	END_CASE
ELSE
	_pulseGenerator(IN := TRUE, PT := T#50MS);	
END_IF
END_METHOD

{attribute 'TcRpcEnable' := '1'}
METHOD RaisePropertiesChanged
VAR_INPUT
	Execute : BOOL;
END_VAR
IF Execute THEN	
	DistanceMsg := ' ';
	IdMsg := ' ';
	CustomMsg := ' ';
END_IF
END_METHOD

END_FUNCTION_BLOCK

// ---- PMShared/Hardware/Devices/DistanceSensors/DistanceSensorBase.TcPOU
FUNCTION_BLOCK ABSTRACT DistanceSensorBase EXTENDS TExecution IMPLEMENTS IDevice
VAR_INPUT
END_VAR
VAR_OUTPUT
END_VAR
VAR
	{attribute 'OPC.UA.DA' := '0'}
	_name : STRING;
	{attribute 'OPC.UA.DA' := '0'}
	_deviceID : STRING;					
	{attribute 'OPC.UA.DA' := '0'}
	_family : DeviceFamily;	
	{attribute 'OPC.UA.DA' := '0'}
	_logger : Logger;
	{attribute 'OPC.UA.DA' := '0'}
	_message : StringBuilder;
	{attribute 'OPC.UA.DA' := '0'}
	_distanceSensorConfig : DeviceConfiguration;
END_VAR

PROPERTY DeviceID : STRING
GET
DeviceID := _deviceID;
END_GET
SET
_deviceID := DeviceID;
END_SET
END_PROPERTY

PROPERTY Family : DeviceFamily
GET
Family := _family;
END_GET
SET
_family := Family;
END_SET
END_PROPERTY

PROPERTY Name : STRING
GET
Name := _name;
END_GET
SET
_name := Name;
END_SET
END_PROPERTY

END_FUNCTION_BLOCK

// ---- PMShared/Hardware/Devices/MPPCs/Hamamatsu/C13336/C13336MppcWide.TcPOU
FUNCTION_BLOCK C13336MppcWide EXTENDS C13336Mppc
VAR_INPUT
END_VAR
VAR_OUTPUT
END_VAR
VAR
	{attribute 'OPC.UA.DA' := '0'}
	_config : C13336MppcConfig;
	
	{attribute 'OPC.UA.DA' := '0'}
	_initDevice : BOOL;
	
	{attribute 'OPC.UA.DA.Access' := '0'}
    InputMppcWideStateSignal_1	AT %I* : BOOL;
	
	{attribute 'OPC.UA.DA.Access' := '0'}
    InputMppcWideStateSignal_2	AT %I* : BOOL;
	
	{attribute 'OPC.UA.DA' := '0'}
	_itemInit : INT;
	{attribute 'OPC.UA.DA' := '0'}
	_pulseGeneratorInit : TON;
	
	{attribute 'OPC.UA.DA' := '0'}
	_coeAccess : CoeAccess;
	{attribute 'OPC.UA.DA' := '0'}
	_initConfigSerialCom : BOOL;
	{attribute 'OPC.UA.DA' := '0'}
	_serialCom  : SerialCom(Prefix := Const.START_OF_TEXT, Suffix := Const.CARRIAGE_RETURN);
	{attribute 'OPC.UA.DA' := '0'}
	_refSerialCom : REFERENCE TO SerialCom(Prefix := Const.START_OF_TEXT, Suffix := Const.CARRIAGE_RETURN) := _serialCom;
		
END_VAR

IF NOT _raiseProperties THEN
	GetStateSignals();
END_IF

// Init device
SUPER^.InitDevice();

IF InitConfigSerialCom AND MppcActivate THEN
	THIS^.Status := TExecutionState.Ready;
ELSE
    THIS^.Status := TExecutionState.Error;	
END_IF

IF THIS^.Status = TExecutionState.Ready THEN
	SUPER^(Conf := _config, SerialCom := _serialCom, RefSerialCom := _refSerialCom);
END_IF

IF SUPER^._initDeviceBase THEN	
	IF NOT InitConfigSerialCom THEN
		ConfigureSerialCom();
	ELSIF THIS^.Status = TExecutionState.Ready THEN						
		_refSerialCom(TxBuffer:= HardwareGlobalVariables.TxBufferMppcWide, 
					  RxBuffer:= HardwareGlobalVariables.RxBufferMppcWide);		

		// Start Mppc to off 
		IF NOT _initDevice THEN
			InitDevice();
		END_IF					
	END_IF
END_IF

METHOD ConfigureSerialCom
VAR_INPUT
END_VAR

VAR
	Status: INT;
END_VAR
IF _coeAccess.CoeOperation.Ready THEN
	_logger.Information(_message.Reset().Append('Start configuration com serial').ToString());
END_IF;	

_coeAccess.CoeOperation.Start();
_coeAccess(SerialCommunication := _config.SerialCommunication);
	
IF _coeAccess.CoeOperation.Done THEN
	_coeAccess.SetDone();
	
	_Logger.Information(_message.Reset().
							Append('{').Append(TO_STRING(THIS^.Family)).Append('} : ').
							Append(' - Status : ').Append(TO_STRING(_coeAccess.Status)).ToString());
	InitConfigSerialCom := TRUE;
END_IF
 
IF _coeAccess.CoeOperation.Error THEN	
	_coeAccess.SetError(0);
	
	_Logger.Error(_message.Reset().
							Append('{').Append(TO_STRING(THIS^.Family)).Append('} : ').
							Append(' - Status : ').Append(TO_STRING(_coeAccess.Status)).ToString());
	InitConfigSerialCom := TRUE;
END_IF

THIS^.Status := _coeAccess.Status;
State := _coeAccess.Status;
END_METHOD

METHOD FB_init : BOOL
VAR_INPUT
	bInitRetains : BOOL; // if TRUE, the retain variables are initialized (warm start / cold start)
	bInCopyCode : BOOL;  // if TRUE, the instance afterwards gets moved into the copy code (online change)
	Config : C13336MppcConfig;
END_VAR
IF Config.IsEnabled THEN
	_config := Config;
	
	SUPER^._mppcConfig.Name := Config.Name;
	SUPER^._mppcConfig.DeviceID := Config.DeviceID;
	SUPER^._mppcConfig.IsEnabled := Config.IsEnabled;
	SUPER^._mppcConfig.LogLevel := Config.LogLevel;
	
	SUPER^.Name := Config.Name;
	SUPER^.DeviceID := Config.DeviceID;	
	THIS^.Family := DeviceFamily.MPPC;
		
	_Logger.Information(_message.Reset().Append('Init ').
							Append('{').Append(TO_STRING(THIS^.Family)).Append('} - ').
							Append('{').Append(TO_STRING(Config.Name)).Append('}').ToString());																													
END_IF
END_METHOD

METHOD GetStateSignals
VAR_INPUT
END_VAR
VAR
	{attribute 'OPC.UA.DA' := '0'}
	fibersCollector : STRING;
	{attribute 'OPC.UA.DA' := '0'}
	delimeter : STRING := ';';
	{attribute 'OPC.UA.DA' := '0'}
	stateSignal : STRING;	
	
END_VAR

fibersCollector := CONCAT(TO_STRING(EMppcCollector.WIDE), delimeter);

IF NOT InputMppcWideStateSignal_1 AND NOT InputMppcWideStateSignal_2 THEN
	stateSignal := CONCAT(fibersCollector, TO_STRING(EMppcStateModule.UNRECOVERABLE_ERROR));
ELSIF NOT InputMppcWideStateSignal_1 AND InputMppcWideStateSignal_2 THEN
	stateSignal := CONCAT(fibersCollector, TO_STRING(EMppcStateModule.AWAITING_COOLING_TEMP_STABLE));
ELSIF InputMppcWideStateSignal_1 AND NOT InputMppcWideStateSignal_2 THEN
	stateSignal := CONCAT(fibersCollector, TO_STRING(EMppcStateModule.AWAITING_HIGH_VOLTAGE_POWER_SUPPLY_STABLE));
ELSE
	stateSignal := CONCAT(fibersCollector, TO_STRING(EMppcStateModule.MODULE_OPERATING_NORMAL));
END_IF

IF stateSignal <> SUPER^.StateSignalsMsg THEN	
	SUPER^.StateSignalsMsg := stateSignal;
	SUPER^.GetStateSignals();
END_IF
END_METHOD

PROPERTY InitConfigSerialCom : BOOL
GET
InitConfigSerialCom := _initConfigSerialCom;
END_GET
SET
_initConfigSerialCom := InitConfigSerialCom;
END_SET
END_PROPERTY

METHOD InitDevice
VAR_INPUT
END_VAR
VAR	
END_VAR
IF NOT _initDevice THEN			
	IF _pulseGeneratorInit.Q THEN
		_pulseGeneratorInit(IN := FALSE, PT := T#10MS);
			
		CASE _itemInit OF
			0:  _logger.Information(_message.Reset().
								Append(_config.Name).
								Append(' - Start to on').ToString());		
				_itemInit := 1;
				
			1:  _outputVoltageOn := TRUE;			
				_initDevice := TRUE;
				_itemInit := 0;
		END_CASE
	ELSE
		_pulseGeneratorInit(IN := TRUE, PT := T#500MS);	
	END_IF
END_IF
END_METHOD

END_FUNCTION_BLOCK

// ---- PMShared/Hardware/Devices/MPPCs/Hamamatsu/C13336Mppc.TcPOU
{attribute 'OPC.UA.DA' := '1'}
FUNCTION_BLOCK C13336Mppc EXTENDS MppcBase
VAR_INPUT	
	{attribute 'OPC.UA.DA' := '0'}
	Conf : C13336MppcConfig;
	{attribute 'OPC.UA.DA' := '0'}
	SerialCom  : SerialCom(Prefix := Const.START_OF_TEXT, Suffix := Const.CARRIAGE_RETURN);
	{attribute 'OPC.UA.DA' := '0'}
	RefSerialCom : REFERENCE TO SerialCom(Prefix := Const.START_OF_TEXT, Suffix := Const.CARRIAGE_RETURN) := SerialCom;
	{attribute 'OPC.UA.DA' := '0'}
	MppcActivate : BOOL;
END_VAR
VAR_OUTPUT	
END_VAR
VAR		
	{attribute 'OPC.UA.DA' := '0'}	 
	_isReceived : BOOL;
	
	{attribute 'OPC.UA.DA' := '0'}
	_deliverMessages : INT;
		
	OutputCurrentMsg : STRING(255);
	OutputVoltageMsg : STRING(255);
	OutputVoltageSettingMsg : STRING(255);
	TemperatureMsg : STRING(255);
	SensorTemperatureMsg : STRING(255);
	PowerFctReadMsg : STRING(255);	
	MonitorInfoStatusMsg : STRING(255);
	HighVoltageStatusMsg : STRING(255);	
	TempCorrectionFactorReadMsg : STRING(255);
	FirmwareMsg : STRING(255);
	IdentifierMsg : STRING(255);
	StateSignalsMsg : STRING(255);
	
	{attribute 'OPC.UA.DA' := '0'}
	VoltageStabilityMsg : STRING(255);
	
	{region 'Commands'}
	
	{attribute 'OPC.UA.DA' := '0'}
	_tempCorrectionFactorSetting : BOOL;
	{attribute 'OPC.UA.DA' := '0'}
	_switchTempCompensationMode : BOOL;
	{attribute 'OPC.UA.DA' := '0'}
	_refVoltageTempSetting : BOOL;
	{attribute 'OPC.UA.DA' := '0'}		  
	_powerFctSetting : BOOL;
	{attribute 'OPC.UA.DA' := '0'}			   
	_outputVoltageOn : BOOL;
	{attribute 'OPC.UA.DA' := '0'}		 
	_outputVoltageOff : BOOL;
	{attribute 'OPC.UA.DA' := '0'}
	_powerReset : BOOL;
	{attribute 'OPC.UA.DA' := '0'}
	_customCmd : BOOL;	
	{attribute 'OPC.UA.DA' := '0'}			  		   
	_raiseProperties : BOOL;
	{attribute 'OPC.UA.DA' := '0'}		  
	_powerFctRead : BOOL;
	{attribute 'OPC.UA.DA' := '0'}	
	_overcurrentProtection : BOOL;
	{attribute 'OPC.UA.DA' := '0'}	
	_outputVoltageControl : BOOL;
	{attribute 'OPC.UA.DA' := '0'}	 
	_tempCompensationMode : BOOL;
	{attribute 'OPC.UA.DA' := '0'}			  
	_manageRelays : BOOL;
	{attribute 'OPC.UA.DA' := '0'}
	_ioRelayActivated : BOOL; 
	{attribute 'OPC.UA.DA' := '0'}
	_setOutputVoltage : BOOL;
				   
	{attribute 'OPC.UA.DA' := '0'}
	_collector : STRING;
	{attribute 'OPC.UA.DA' := '0'}
	_fibersCollector : STRING;
	{attribute 'OPC.UA.DA' := '0'}
	_delimeter : STRING := ';';
		 
	{endregion}
		 
	{attribute 'OPC.UA.DA' := '0'}
	_initDeviceBase : BOOL;	
	 
	{attribute 'OPC.UA.DA' := '0'}
	_cmd : STRING;	
	{attribute 'OPC.UA.DA' := '0'}	
	_setRefVoltage : LREAL := 0;
	{attribute 'OPC.UA.DA' := '0'}	
	_setVoltage : LREAL := 0;				
	{attribute 'OPC.UA.DA' := '0'}
	_itemScheduler : INT;		
	{attribute 'OPC.UA.DA' := '0'}
	_itemExecScheduler : INT;
	{attribute 'OPC.UA.DA' := '0'}
	_itemRaisedProperties : INT;
	{attribute 'OPC.UA.DA' := '0'}
	_pulseGenerator : TON;	
			
	{attribute 'OPC.UA.DA' := '0'}
	message : STRING;
	{attribute 'OPC.UA.DA' := '0'}
	tmpMessage : STRING;
	
	{attribute 'OPC.UA.DA' := '0'}
	msgWithoutPrefix : STRING;
	{attribute 'OPC.UA.DA' := '0'}
	suffixDelete : INT := 5;
	{attribute 'OPC.UA.DA' := '0'}
	prefixDelete : INT := 3;
	
	{attribute 'OPC.UA.DA' := '0'}
	_length : INT;
	{attribute 'OPC.UA.DA' := '0'}
	_conv : BOOL;
	{attribute 'OPC.UA.DA' := '0'}
	valConvert : LREAL;		
	
	
	{attribute 'OPC.UA.DA' := '0'}
	strTmp : STRING;
	{attribute 'OPC.UA.DA' := '0'}
	strTmp1 : STRING;
	
END_VAR

IF SerialCom.ErrorSendId <> COMERROR_NOERROR THEN
	RETURN;
END_IF

// Deliver messages
IF RefSerialCom.IsReceived THEN
	IF (Conf.DeviceID = TO_STRING(EMppcCollector.WIDE)) THEN
		_collector := TO_STRING(EMppcCollector.WIDE);
	ELSE
		_collector := TO_STRING(EMppcCollector.NARROW);
	END_IF	
		
	_fibersCollector := CONCAT(_collector, _delimeter);
	
	msgWithoutPrefix := DELETE(RefSerialCom.LastReceivedString, suffixDelete, 0);	
	_length := LEN(msgWithoutPrefix);
	message := DELETE(msgWithoutPrefix, _length - prefixDelete, _length - prefixDelete);

	CASE _deliverMessages OF		
		EFeedbackMsgC13336.MonitorInfoStatusMsg :
		 	MonitorInfoStatusMsg := CONCAT(_fibersCollector, message); 
			VoltageStabilityMsg := CONCAT(_fibersCollector, FindVoltageStability(message)); 
			HighVoltageStatusMsg := CONCAT(_fibersCollector, FindHighVoltageOutput(message));
			
		EFeedbackMsgC13336.OutputCurrentMsg :			
			OutputCurrentMsg := CONCAT(_fibersCollector, ConvertMonitorHexaToCurrent(message));	
			
		EFeedbackMsgC13336.OutputVoltageMsg :
			OutputVoltageMsg := CONCAT(_fibersCollector, ConvertMonitorHexaToVoltage(message));	
			
		EFeedbackMsgC13336.OutputVoltageSettingMsg :			
			tmpMessage := LEFT(RIGHT(message, 8), 4);		
			OutputVoltageSettingMsg := CONCAT(_fibersCollector, ConvertMonitorHexaToVoltage(tmpMessage));		
	
		EFeedbackMsgC13336.TemperatureMsg :
			TemperatureMsg := CONCAT(_fibersCollector, message);
			
		EFeedbackMsgC13336.SensorTemperatureMsg :
			tmpMessage := LEFT(RIGHT(message, 8), 4);
			SensorTemperatureMsg := CONCAT(_fibersCollector, ConvertMonitorHexaToTemperature(tmpMessage));
	
		EFeedbackMsgC13336.PowerFctReadMsg :
			PowerFctReadMsg := CONCAT(_fibersCollector, message);
			
		EFeedbackMsgC13336.TempCorrectionFactorReadMsg :
			TempCorrectionFactorReadMsg := CONCAT(_fibersCollector, message);

		EFeedbackMsgC13336.FirmwareMsg :
			FirmwareMsg := CONCAT(_fibersCollector, message);	
			
		EFeedbackMsgC13336.IdentifierMsg :
			IdentifierMsg := CONCAT(_fibersCollector, message);					
	END_CASE	
END_IF						   							   		
	
TempCorrectionFactorSetting(_tempCorrectionFactorSetting);
SwitchTempCompensationMode(_switchTempCompensationMode, _tempCompensationMode);
RefVoltageTempSetting(_refVoltageTempSetting, _setRefVoltage);
PowerFctSetting(_powerFctSetting, _overcurrentProtection, _outputVoltageControl);
OutputVoltageOn(_outputVoltageOn);
OutputVoltageOff(_outputVoltageOff);
PowerReset(_powerReset);
CustomCommand(_customCmd, _cmd);
RaisePropertiesChanged(_raiseProperties);		
ManageRelays(_manageRelays, _ioRelayActivated);
SetOutputVoltage(_setOutputVoltage, _setVoltage);


IF (NOT _tempCorrectionFactorSetting AND NOT _switchTempCompensationMode AND NOT _refVoltageTempSetting AND NOT _powerFctSetting AND
	NOT _outputVoltageOn AND NOT _outputVoltageOff AND NOT _powerReset AND NOT _raiseProperties AND NOT _manageRelays) THEN
	
	MessageScheduler();	
END_IF

(** Convert Hexa to mA **)
METHOD ConvertMonitorHexaToCurrent : STRING
VAR_INPUT
	Data : STRING;	
END_VAR
VAR
	dataInDec : STRING;
	dataToDint : DINT;
END_VAR
dataInDec := CONCAT('16#', Data);
dataToDint := STRING_TO_DINT(dataInDec);
ConvertMonitorHexaToCurrent := LREAL_TO_FMTSTR(DINT_TO_LREAL(dataToDint) * 0.005194, 3, TRUE);
END_METHOD

(** Convert Hexa to Temperature **)
METHOD ConvertMonitorHexaToTemperature : STRING
VAR_INPUT
	Data : STRING;
END_VAR
VAR
	dataInDec : STRING;
	dataToDint : DINT;
	
	sTmp0 : STRING;
	sTmp1 : STRING;
	sTmp2 : STRING;
	sTemperature : STRING;
END_VAR
dataInDec := CONCAT('16#', Data);
dataToDint := STRING_TO_DINT(dataInDec);

IF dataToDint > 0 THEN
	sTmp0 := LREAL_TO_FMTSTR((DINT_TO_LREAL(dataToDint) * 10000.0) / (1024.0 - DINT_TO_LREAL(dataToDint)) * (1 / 9000.0), 15, FALSE);
	IF STRING_TO_LREAL(sTmp0) > 0 THEN		
		sTmp1 := LREAL_TO_FMTSTR(LN(STRING_TO_LREAL(sTmp0)), 15, FALSE);
		sTmp2 := LREAL_TO_FMTSTR(STRING_TO_LREAL(sTmp1) * (1 / 3410.0) + (1 / 298.15), 15, FALSE);
		sTemperature := LREAL_TO_FMTSTR(1 / STRING_TO_LREAL(sTmp2) - 273.15, 3, FALSE);
	ELSE
		sTemperature := 'NaN';
	END_IF
ELSE
	sTemperature := 'NaN';

END_IF

ConvertMonitorHexaToTemperature := sTemperature;
END_METHOD

(** Convert Hexa to Volt **)
METHOD ConvertMonitorHexaToVoltage : STRING
VAR_INPUT
	Data : STRING;
END_VAR
VAR
	dataInDec : STRING;
	dataToDint : DINT;
END_VAR
dataInDec := CONCAT('16#', Data);
dataToDint := STRING_TO_DINT(dataInDec);
ConvertMonitorHexaToVoltage := LREAL_TO_FMTSTR(DINT_TO_LREAL(dataToDint) * 0.001812, 3, TRUE);
END_METHOD

METHOD ConvertMonitorVoltageToHexa : ARRAY[0..3] OF STRING
VAR_INPUT
	Data : LREAL;
END_VAR
VAR
	dataCoef : STRING;
	dataToDWord : DWORD;	
	
	sMonitorVoltageToHex : STRING;	
	arrayVoltageToHex : ARRAY[0..3] OF STRING;
	
	counter : INT;
	iLenVoltage : INT;
	
	lTmp1 : LREAL;
	lTmp2 : LREAL;
	
	sTmp1 : STRING;
END_VAR
lTmp1 := Data / 0.001812;
lTmp2 := FRAC(lTmp1);
IF lTmp2 < 0.5 THEN
	dataCoef := LREAL_TO_STRING(lTmp1);
ELSE
	dataCoef := LREAL_TO_STRING(lTmp1 + 1);
END_IF

dataToDWord := STRING_TO_DWORD(dataCoef);
sMonitorVoltageToHex := DWORD_TO_HEXSTR(dataToDWord, 4, FALSE);

iLenVoltage := LEN(sMonitorVoltageToHex);
FOR counter := 0 TO iLenVoltage - 1 BY 1 DO
	sTmp1 := MID(sMonitorVoltageToHex, 1, counter + 1);
	arrayVoltageToHex[counter] := BYTE_TO_HEXSTR(F_ToASC(sTmp1), 1, FALSE);
END_FOR;

ConvertMonitorVoltageToHexa := arrayVoltageToHex;
END_METHOD

METHOD ConvertStatusMessage : STRING
VAR_INPUT
	Status : STRING;
END_VAR
VAR
	voltageOutputMessage : BOOL;

	tmp : UINT;		
END_VAR
tmp := STRING_TO_UINT(RIGHT(Status, 1));

voltageOutputMessage := UINT_TO_BOOL(tmp);

IF voltageOutputMessage THEN
	ConvertStatusMessage := 'ON'; 	
ELSE
	ConvertStatusMessage := 'OFF';
END_IF
END_METHOD

{attribute 'TcRpcEnable' := '1'}
(** Custom command **)
METHOD CustomCommand 
VAR_INPUT
	Execute : BOOL;
	Cmd : STRING;
END_VAR
IF Execute THEN
	_logger.Information(_message.Reset().
								Append(Conf.Name).
								Append(' - Custom command : ').
								Append(Cmd).ToString());	
	_deliverMessages := EFeedbackMsgC13336.CustomMsg;														
	SerialCom.Send(Cmd);	
	_customCmd := FALSE;
END_IF
END_METHOD

METHOD FindHighVoltageOutput : STRING
VAR_INPUT
	message : STRING;
END_VAR
VAR
	{attribute 'OPC.UA.DA' := '0'}	
	_monitorHighVoltageStatus : STRING(255);			
	{attribute 'OPC.UA.DA' := '0'}
	statusMessageBin : STRING;
	{attribute 'OPC.UA.DA' := '0'}
	messageToBin : STRING;
	{attribute 'OPC.UA.DA' := '0'}		
	mask : STRING := '16#1';
	{attribute 'OPC.UA.DA' := '0'}
	status : WORD;
	{attribute 'OPC.UA.DA' := '0'}
	statusMsg : WORD;
END_VAR
statusMsg := STRING_TO_WORD(CONCAT('16#', LEFT(message, 4)));
statusMessageBin := WORD_TO_BINSTR(statusMsg, 16);

status := STRING_TO_WORD(statusMessageBin) AND STRING_TO_WORD(mask);

IF status = 0 THEN
	_monitorHighVoltageStatus := 'OFF';
ELSE
	_monitorHighVoltageStatus := 'ON';
END_IF

FindHighVoltageOutput := _monitorHighVoltageStatus;
END_METHOD

METHOD FindVoltageStability : STRING
VAR_INPUT
	message : STRING;
END_VAR
VAR
	{attribute 'OPC.UA.DA' := '0'}	
	_monitorInfoStatus : STRING(255);		
	{attribute 'OPC.UA.DA' := '0'}
	one : WORD := 1;
	{attribute 'OPC.UA.DA' := '0'}
	isolStatus : DWORD;
	{attribute 'OPC.UA.DA' := '0'}
	statusMessageBin : STRING;
	{attribute 'OPC.UA.DA' := '0'}
	messageToBin : STRING;
	{attribute 'OPC.UA.DA' := '0'}
	valueStatus : WORD;
	{attribute 'OPC.UA.DA' := '0'}		
	mask : STRING := '16#4000';
	{attribute 'OPC.UA.DA' := '0'}
	status : WORD;
	{attribute 'OPC.UA.DA' := '0'}
	statusMsg : WORD;
	
END_VAR

statusMsg := STRING_TO_WORD(CONCAT('16#', LEFT(message, 4)));
statusMessageBin := WORD_TO_BINSTR(statusMsg, 16);

status := STRING_TO_WORD(statusMessageBin) AND STRING_TO_WORD(mask);
valueStatus := SHR(status, 14);


IF valueStatus = 0 THEN
	_monitorInfoStatus := 'Unstable';
ELSE
	_monitorInfoStatus := 'Stable';
END_IF

FindVoltageStability := _monitorInfoStatus;
END_METHOD

METHOD GetFirmware
VAR_INPUT
END_VAR
VAR
	// 'HFI'
	cmdArray : ARRAY[0..7] OF BYTE := [16#02, 16#48, 16#46, 16#49, 16#03, 16#44, 16#43, 16#0D];
END_VAR
_deliverMessages := EFeedbackMsgC13336.FirmwareMsg;
SerialCom.Send8B(cmdArray);
END_METHOD

METHOD GetIdentifier
VAR_INPUT
END_VAR
VAR
	// 'HGN'
	cmdArray : ARRAY[0..7] OF BYTE := [16#02, 16#48, 16#47, 16#4F, 16#03, 16#45, 16#32, 16#0D]; 
END_VAR
 _deliverMessages := EFeedbackMsgC13336.IdentifierMsg;
SerialCom.Send8B(cmdArray);
END_METHOD

METHOD GetMonitorInfoStatus
VAR_INPUT
END_VAR
VAR
	// 'HPO'
	cmdArray : ARRAY[0..7] OF BYTE := [16#02, 16#48, 16#50, 16#4F, 16#03, 16#45, 16#43, 16#0D];
END_VAR
_deliverMessages := EFeedbackMsgC13336.MonitorInfoStatusMsg;
SerialCom.Send8B(cmdArray);
END_METHOD

METHOD GetOutputCurrent
VAR_INPUT
END_VAR
VAR
	// 'HGC'
	cmdArray : ARRAY[0..7] OF BYTE := [16#02, 16#48, 16#47, 16#43, 16#03, 16#44, 16#37, 16#0D]; 
END_VAR
_deliverMessages := EFeedbackMsgC13336.OutputCurrentMsg;
SerialCom.Send8B(cmdArray);
END_METHOD

METHOD GetOutputVoltage
VAR_INPUT
END_VAR
VAR
	// 'HGV'
	cmdArray : ARRAY[0..7] OF BYTE := [16#02, 16#48, 16#47, 16#56, 16#03, 16#45, 16#41, 16#0D]; 
END_VAR
_deliverMessages := EFeedbackMsgC13336.OutputVoltageMsg;
SerialCom.Send8B(cmdArray);
END_METHOD

METHOD GetOutputVoltageSetting
VAR_INPUT
END_VAR
VAR
	// 'HRT'
	cmdArray : ARRAY[0..7] OF BYTE := [16#02, 16#48, 16#52, 16#54, 16#03, 16#46, 16#33, 16#0D]; 
END_VAR
_deliverMessages := EFeedbackMsgC13336.OutputVoltageSettingMsg;
SerialCom.Send8B(cmdArray);
END_METHOD

METHOD GetSensorTemperature
VAR_INPUT
END_VAR
VAR
	// 'TGV'
	cmdArray : ARRAY[0..7] OF BYTE := [16#02, 16#54, 16#47, 16#56, 16#03, 16#46, 16#36, 16#0D]; 
END_VAR
_deliverMessages := EFeedbackMsgC13336.SensorTemperatureMsg;
SerialCom.Send8B(cmdArray);
END_METHOD

METHOD GetStateSignals
VAR_INPUT
END_VAR
_deliverMessages := EFeedbackMsgC13336.StateSignalsMsg;
END_METHOD

METHOD GetStatus
VAR
	// 'HGS'
	cmdArray : ARRAY[0..7] OF BYTE := [16#02, 16#48, 16#47, 16#53, 16#03, 16#45, 16#37, 16#0D]; 
END_VAR
_deliverMessages := EFeedbackMsgC13336.StatusMsg;
SerialCom.Send8B(cmdArray);
END_METHOD

METHOD GetTemperature
VAR_INPUT
END_VAR
VAR
	// 'HGT'
	cmdArray : ARRAY[0..7] OF BYTE := [16#02, 16#48, 16#47, 16#54, 16#03, 16#45, 16#38, 16#0D]; 
END_VAR
_deliverMessages := EFeedbackMsgC13336.TemperatureMsg;
SerialCom.Send8B(cmdArray);
END_METHOD

METHOD InitDevice
VAR_INPUT
END_VAR
IF NOT _initDeviceBase THEN	
	_logger.Information(_message.Reset().
								Append(Conf.Name).
								Append(' - Activates relays').ToString());
		
	ManageRelays(TRUE, TRUE);			
	_initDeviceBase := TRUE;	
END_IF
END_METHOD

METHOD ManageRelays
VAR_INPUT
	Execute : BOOL;
	IoRelay : BOOL;
END_VAR
IF Execute THEN
	_logger.Information(_message.Reset().
								Append('MPPCs relay: ').
								Append(BOOL_TO_STRING(IoRelay)).ToString());	

	// Physically activates relay			
	MppcActivate := IoRelay;
	
	_manageRelays := FALSE;
END_IF
END_METHOD

METHOD MessageScheduler
VAR_INPUT
END_VAR
IF _pulseGenerator.Q THEN
	_pulseGenerator(IN := FALSE, PT := T#10MS);
		
	CASE _itemScheduler OF		
		0: GetOutputCurrent();
			_itemScheduler := 1;
				
		1: GetOutputVoltage();
			_itemScheduler := 2;
			
		2: GetMonitorInfoStatus();
			_itemScheduler := 3;
			
		3: GetSensorTemperature();
			_itemScheduler := 0;
	END_CASE
ELSE
	_pulseGenerator(IN := TRUE, PT := T#200MS);	
END_IF
END_METHOD

{attribute 'TcRpcEnable' := '1'}
METHOD OutputVoltageOff
VAR_INPUT
	Execute : BOOL;
END_VAR
VAR	
	// 'HOF'
	cmdArray : ARRAY[0..7] OF BYTE := [16#02, 16#48, 16#4F, 16#46, 16#03, 16#45, 16#32, 16#0D]; 
END_VAR
IF Execute THEN		
	_outputVoltageOff := TRUE;
	
	IF _pulseGenerator.Q THEN
		_pulseGenerator(IN := FALSE, PT := T#10MS);
		
		CASE _itemExecScheduler OF		
			0:  _logger.Information(_message.Reset().
								Append(Conf.Name).
								Append(' - OutputVoltageOff').ToString());
				SerialCom.Send8B(cmdArray);   
				_itemExecScheduler := 1;
				
			1: GetStatus(); 
				_outputVoltageOff := FALSE;
				_itemExecScheduler := 0;
		
		END_CASE	
	ELSE
		_pulseGenerator(IN := TRUE, PT := T#200MS);	
	END_IF									
END_IF
END_METHOD

{attribute 'TcRpcEnable' := '1'}
METHOD OutputVoltageOn
VAR_INPUT
	Execute : BOOL;
END_VAR
VAR
	// 'HON'
	cmdArray : ARRAY[0..7] OF BYTE := [16#02, 16#48, 16#4F, 16#4E, 16#03, 16#45, 16#41, 16#0D]; 
END_VAR
IF Execute THEN		
	_outputVoltageOn := TRUE;
	
	IF _pulseGenerator.Q THEN
		_pulseGenerator(IN := FALSE, PT := T#10MS);
		
		CASE _itemExecScheduler OF		
			0:  _logger.Information(_message.Reset().
								Append(Conf.Name).
								Append(' - OutputVoltageOn').ToString());
				SerialCom.Send8B(cmdArray);   
				_itemExecScheduler := 0;
				_outputVoltageOn := FALSE;
				
			1: GetStatus(); 
				_outputVoltageOn := FALSE;
				_itemExecScheduler := 0;
		
		END_CASE	
	ELSE
		_pulseGenerator(IN := TRUE, PT := T#2000MS);	
	END_IF									
END_IF
END_METHOD

METHOD PowerFctRead
VAR_INPUT	
END_VAR
VAR
	// 'HRC'
	cmdArray : ARRAY[0..7] OF BYTE := [16#02, 16#48, 16#52, 16#43, 16#03, 16#45, 16#32, 16#0D]; 
END_VAR
_deliverMessages := EFeedbackMsgC13336.PowerFctReadMSg;
SerialCom.Send8B(cmdArray);
END_METHOD

{attribute 'TcRpcEnable' := '1'}
METHOD PowerFctSetting
VAR_INPUT
	Execute : BOOL;
	OvercurrentProtection : BOOL;
	OutputVoltageControl : BOOL;
END_VAR
VAR
	// 'HSC'
	cmdArray : ARRAY[0..11] OF BYTE; 
	data : BYTE := 16#32;
	checksum : BYTE;
END_VAR
IF Execute THEN
	_logger.Information(_message.Reset().
								Append(Conf.Name).
								Append(' - PowerFctSetting').ToString());		

	IF OvercurrentProtection AND OutputVoltageControl THEN 
		data := 16#33;
		checksum := 16#36;
	ELSIF OvercurrentProtection AND NOT OutputVoltageControl THEN
		data := 16#31;
		checksum := 16#34;
	ELSIF NOT OvercurrentProtection AND OutputVoltageControl THEN
		data := 16#32;
		checksum := 16#35;
	ELSE
		data := 16#30;
		checksum := 16#33;	
	END_IF	
	
	cmdArray[0] := 16#02;
	cmdArray[1] := 16#48; 
	cmdArray[2] := 16#53; 
	cmdArray[3] := 16#43; 
	cmdArray[4] := 16#30; 
	cmdArray[5] := 16#30; 
	cmdArray[6] := 16#30; 
	cmdArray[7] := data;	
	cmdArray[8] := 16#03; 
	cmdArray[9] := 16#41; 
	cmdArray[10] := checksum; 
	cmdArray[11] := 16#0D; 
										
	SerialCom.Send12B(cmdArray);
	_powerFctSetting := FALSE;
END_IF
END_METHOD

{attribute 'TcRpcEnable' := '1'}
METHOD PowerReset
VAR_INPUT
	Execute : BOOL;
END_VAR
VAR
	// 'HRE'
	cmdArray : ARRAY[0..7] OF BYTE := [16#02, 16#48, 16#52, 16#45, 16#03, 16#45, 16#34, 16#0D]; 
END_VAR
IF Execute THEN		
	_powerReset := TRUE;
	
	IF _pulseGenerator.Q THEN
		_pulseGenerator(IN := FALSE, PT := T#10MS);
		
		CASE _itemExecScheduler OF		
			0:  _logger.Information(_message.Reset().
								Append(Conf.Name).
								Append(' - PowerReset').ToString());
				SerialCom.Send8B(cmdArray);   
				_itemExecScheduler := 2;				
				
			1: GetStatus(); 
				_itemExecScheduler := 2;
				
			2:	_powerReset := FALSE;
				_itemExecScheduler := 0;
		
		END_CASE	
	ELSE
		_pulseGenerator(IN := TRUE, PT := T#500MS);	
	END_IF									
END_IF
END_METHOD

{attribute 'TcRpcEnable' := '1'}
METHOD RaisePropertiesChanged
VAR_INPUT
	Execute : BOOL;
END_VAR

(*
Ajouter fonction pour remonter les états des 2 IOs quand C# en fait la demande.
La même chose avec LE On/off où l'info n'est pas remontée vu qu'elle n'a pas changé
*)
IF Execute THEN	
	_raiseProperties := TRUE;
	
	IF _pulseGenerator.Q THEN
		_pulseGenerator(IN := FALSE, PT := T#10MS);
	
		CASE _itemRaisedProperties OF		
			0:  //OutputCurrentMsg := ' ';	
				//OutputVoltageMsg := ' ';			    		   			    		   
			    //SensorTemperatureMsg := ' ';			    
				OutputVoltageSettingMsg := ' ';	
			    StateSignalsMsg := ' ';	
			    			    
			    TemperatureMsg := ' ';
			    FirmwareMsg := ' ';
			    TempCorrectionFactorReadMsg := ' ';				   
   			    HighVoltageStatusMsg := ' ';	
                IdentifierMsg := ' ';
			    PowerFctReadMsg := ' ';		   
			   
				_itemRaisedProperties := 10;													

			10:  GetOutputVoltageSetting();
				_itemRaisedProperties := 11;			
				
			11: GetStateSignals();
				_itemRaisedProperties := 12;
								
			12: _logger.Information(_message.Reset().Append(Conf.Name).
													 Append(' - RaisePropertiesChanged').ToString());
				_raiseProperties := FALSE;
				_itemRaisedProperties := 0;
				
			(* Not necessary for the moment *)			
			30: GetOutputCurrent();
				_itemRaisedProperties := 31;

			31: GetOutputVoltage();
				_itemRaisedProperties := 32;						
																				
			32: GetSensorTemperature();
				_itemRaisedProperties := 33;
			
			33: GetMonitorInfoStatus();
				_itemRaisedProperties := 34;
								
			34: GetFirmware();
				_itemRaisedProperties := 35;
				
			35: TempCorrectionFactorRead();
				_itemRaisedProperties := 36;
				
			36: GetTemperature();
				_itemRaisedProperties := 37;
				
			37: PowerFctRead();
				_itemRaisedProperties := 38;
				
			38: GetIdentifier();
				_itemRaisedProperties := 0;
									
		END_CASE
	
	ELSE
		_pulseGenerator(IN := TRUE, PT := T#500MS);	
	END_IF
END_IF
END_METHOD

{attribute 'TcRpcEnable' := '1'}
METHOD RefVoltageTempSetting
VAR_INPUT
	Execute    : BOOL;
	RefVoltage : LREAL;
END_VAR
VAR
	convertToString : STRING;

	refVoltatgeToArray : ARRAY[0..3] OF STRING; 	

	// 'HBV'
	cmdArray : ARRAY[0..11] OF BYTE; // := [2, 48, 66, 86, 55, 53, 69, 66, 3, 50, 67, 13];
END_VAR
IF Execute THEN
	_logger.Information(_message.Reset().
								Append(Conf.Name).
								Append(' - RefVoltageTempSetting').ToString());	

	refVoltatgeToArray := ConvertMonitorVoltageToHexa(RefVoltage);	

	cmdArray[0] := 16#02;
	cmdArray[1] := 16#30; //48;
	cmdArray[2] := 16#42; //66;
	cmdArray[3] := 16#56; //86;	
	cmdArray[4] := STRING_TO_BYTE(refVoltatgeToArray[0]);
	cmdArray[5] := STRING_TO_BYTE(refVoltatgeToArray[1]);
	cmdArray[6] := STRING_TO_BYTE(refVoltatgeToArray[2]);
	cmdArray[7] := STRING_TO_BYTE(refVoltatgeToArray[3]);	
	cmdArray[8] :=16#03;
	cmdArray[9] := 16#32; //50;
	cmdArray[10] := 16#43; //67;
	cmdArray[11] := 16#0D; //13;
				
	SerialCom.Send12B(cmdArray);
	_refVoltageTempSetting := FALSE;
END_IF
END_METHOD

{attribute 'TcRpcEnable' := '1'}
METHOD SetOutputVoltage
VAR_INPUT
	Execute : BOOL;
	SetVoltage : LREAL;
END_VAR
VAR
	convertToString : STRING;
	setVoltatgeToArrayToHex : ARRAY[0..3] OF STRING; 	

	// 'HST'
	cmdArray : ARRAY[0..31] OF BYTE; 
	
	voltageChecksum : DINT;
	counter : INT;
	
	sPartOfChecksum : STRING := '16#4B4'; // Part of checksum, without voltage value (in hex)	
	wSumVoltageValueToHex : WORD;
	wChecksumTotalToDec : WORD;
	sChecksumTotalToHex : STRING;
	ArrayChecksum : ARRAY[0..MAX_STRING_LENGTH] OF BYTE;
	
	iLenCheksum : INT;
	lastByteChecksum : BYTE;
	secondLastByteChecksum : BYTE;
	
	sLastByteChecksum : STRING;
	sSecondLastByteChecksum : STRING;	
	
	sLastByteChecksumHex : STRING;
	sSecondLastByteChecksumHex : STRING;
	
END_VAR
IF Execute THEN
	_logger.Information(_message.Reset().
								Append(Conf.Name).
								Append(' - Set Output Voltage').ToString());	

	setVoltatgeToArrayToHex := ConvertMonitorVoltageToHexa(SetVoltage);	

	(** Checksum **)
	// Add voltage value and convert it to decimal  
	FOR counter := 0 TO 3 BY 1 DO
		IF counter = 0 THEN
			wSumVoltageValueToHex := STRING_TO_WORD(CONCAT('16#', setVoltatgeToArrayToHex[counter]));
		ELSE
			wSumVoltageValueToHex := wSumVoltageValueToHex + STRING_TO_WORD(CONCAT('16#', setVoltatgeToArrayToHex[counter]));	
		END_IF					
	END_FOR;	
	
	wChecksumTotalToDec := STRING_TO_WORD(sPartOfChecksum) + wSumVoltageValueToHex;
	sChecksumTotalToHex := DWORD_TO_HEXSTR(wChecksumTotalToDec, 1, FALSE);		
	
	ArrayChecksum := MAXSTRING_TO_BYTEARR(sChecksumTotalToHex);
	iLenCheksum := LEN(sChecksumTotalToHex);	
	
	sSecondLastByteChecksum := MID(sChecksumTotalToHex, 1, iLenCheksum-1);
	sSecondLastByteChecksumHex := BYTE_TO_HEXSTR(F_ToASC(sSecondLastByteChecksum), 1, FALSE);
	sLastByteChecksum := MID(sChecksumTotalToHex, 1, iLenCheksum);	
	sLastByteChecksum :=  BYTE_TO_HEXSTR(F_ToASC(sLastByteChecksum), 1, FALSE);
		
	cmdArray[0] := 16#02;
	cmdArray[1] := 16#48; //72;
	cmdArray[2] := 16#53; //83;
	cmdArray[3] := 16#54; //84;
	cmdArray[4] := 16#30; //48;
	cmdArray[5] := 16#30; //48;
	cmdArray[6] := 16#30; //48;
	cmdArray[7] := 16#30; //48;
	cmdArray[8] := 16#30; //48;
	cmdArray[9] := 16#30; //48;
	cmdArray[10] := 16#30; //48;
	cmdArray[11] := 16#30; //48;
	cmdArray[12] := 16#30; //48;
	cmdArray[13] := 16#30; //48;
	cmdArray[14] := 16#30; //48;
	cmdArray[15] := 16#30; //48;
	cmdArray[16] := 16#30; //48;
	cmdArray[17] := 16#30; //48;
	cmdArray[18] := 16#30; //48;
	cmdArray[19] := 16#30; //48;	
	cmdArray[20] := STRING_TO_BYTE(CONCAT('16#', setVoltatgeToArrayToHex[0]));
	cmdArray[21] := STRING_TO_BYTE(CONCAT('16#', setVoltatgeToArrayToHex[1]));
	cmdArray[22] := STRING_TO_BYTE(CONCAT('16#', setVoltatgeToArrayToHex[2]));
	cmdArray[23] := STRING_TO_BYTE(CONCAT('16#', setVoltatgeToArrayToHex[3]));
	cmdArray[24] := 16#30; //48;
	cmdArray[25] := 16#30; //48;
	cmdArray[26] := 16#30; //48;
	cmdArray[27] := 16#30; //48;		
	cmdArray[28] := 16#03;
	cmdArray[29] := STRING_TO_BYTE(CONCAT('16#', sSecondLastByteChecksumHex)); // 16#38 -> 56;
	cmdArray[30] := STRING_TO_BYTE(CONCAT('16#', slastByteChecksum)); // 16#42 -> 66;
	cmdArray[31] := 16#0D; //13;
				
	SerialCom.Send32B(cmdArray);
	_setOutputVoltage := FALSE;
END_IF
END_METHOD

{attribute 'TcRpcEnable' := '1'}
METHOD SwitchTempCompensationMode
VAR_INPUT
	Execute : BOOL;
	TempCompensationMode : BOOL; //0: Disable, 1: Enable
END_VAR
VAR
	// 'HCM'
	cmdArray : ARRAY[0..8] OF BYTE; 
	compensationMode : BYTE;
	mode : STRING;
END_VAR
IF Execute THEN
	IF TempCompensationMode THEN
		compensationMode := 49;
		mode := 'Enable';
	ELSE
		compensationMode := 48;
		mode := 'Disable';
	END_IF	
	
	_logger.Information(_message.Reset().Append(Conf.Name).
										 Append(' - SwitchTempCompensationMode: ').
										 Append(mode).ToString());
	
	cmdArray[0] := 16#02;
	cmdArray[1] := 16#48;//72;
	cmdArray[2] := 16#43;//67;
	cmdArray[3] := 16#4D;//77;	
	cmdArray[4] := compensationMode;
	cmdArray[5] := 16#03;
	cmdArray[6] := 16#30;//48;
	cmdArray[7] := 16#45;//69;	
	cmdArray[8] := 16#0D;//13;
							
	SerialCom.Send9B(cmdArray);
	_switchTempCompensationMode := FALSE;
END_IF
END_METHOD

METHOD TempCorrectionFactorRead
VAR_INPUT
END_VAR
VAR
	// 'HRT'
	cmdArray : ARRAY[0..7] OF BYTE := [16#02, 16#30, 16#52, 16#54, 16#03, 16#46, 16#33, 16#0D];
END_VAR
_deliverMessages := EFeedbackMsgC13336.TempCorrectionFactorReadMsg;
SerialCom.Send8B(cmdArray);
END_METHOD

{attribute 'TcRpcEnable' := '1'}
METHOD TempCorrectionFactorSetting
VAR_INPUT
	Execute : BOOL;
END_VAR
VAR
	// 'HST'
	cmdArray : ARRAY[0..7] OF BYTE := [16#02, 16#30, 16#53, 16#54, 16#03, 16#46, 16#34, 16#0D];
END_VAR
IF Execute THEN
	_logger.Information(_message.Reset().
								Append(Conf.Name).
								Append(' - TempCorrectionFactorSetting').ToString());								
	SerialCom.Send8B(cmdArray);
	_tempCorrectionFactorSetting := FALSE;
END_IF
END_METHOD

END_FUNCTION_BLOCK

// ---- PMShared/Hardware/Devices/MPPCs/MppcBase.TcPOU
FUNCTION_BLOCK ABSTRACT MppcBase EXTENDS TExecution IMPLEMENTS IDevice
VAR_INPUT
END_VAR
VAR_OUTPUT
END_VAR
VAR
	{attribute 'OPC.UA.DA' := '0'}
	_name : STRING;
	{attribute 'OPC.UA.DA' := '0'}
	_deviceID : STRING;					
	{attribute 'OPC.UA.DA' := '0'}
	_family : DeviceFamily;	
	{attribute 'OPC.UA.DA' := '0'}	
	_logger : Logger;
	{attribute 'OPC.UA.DA' := '0'}
	_message : StringBuilder;
	{attribute 'OPC.UA.DA' := '0'}
	_mppcConfig : DeviceConfiguration;
	

END_VAR

PROPERTY DeviceID : STRING
GET
DeviceID := _deviceID;
END_GET
SET
_deviceID := DeviceID;
END_SET
END_PROPERTY

PROPERTY Family : DeviceFamily
GET
Family := _family;
END_GET
SET
_family := Family;
END_SET
END_PROPERTY

PROPERTY Name : STRING
GET
Name := _name;
END_GET
SET
_name := Name;
END_SET
END_PROPERTY

END_FUNCTION_BLOCK

// ---- PMShared/Hardware/Devices/MPPCs/Hamamatsu/C13336/C13366MppcNarrow.TcPOU
FUNCTION_BLOCK C13366MppcNarrow EXTENDS C13336Mppc
VAR_INPUT
END_VAR
VAR_OUTPUT
END_VAR
VAR
	{attribute 'OPC.UA.DA' := '0'}
	_config : C13336MppcConfig;
	
	{attribute 'OPC.UA.DA' := '0'}
	_initDevice : BOOL;
	
	{attribute 'OPC.UA.DA.Access' := '0'}
    InputMppcNarrowStateSignal_1	AT %I* : BOOL;
	
	{attribute 'OPC.UA.DA.Access' := '0'}
    InputMppcNarrowStateSignal_2	AT %I* : BOOL;
	
	{attribute 'OPC.UA.DA' := '0'}
	_itemInit : INT;
	{attribute 'OPC.UA.DA' := '0'}
	_pulseGeneratorInit : TON;
	
	{attribute 'OPC.UA.DA' := '0'}
	_coeAccess : CoeAccess;
	{attribute 'OPC.UA.DA' := '0'}
	_initConfigSerialCom : BOOL;
	{attribute 'OPC.UA.DA' := '0'}
	_serialCom  : SerialCom(Prefix := Const.START_OF_TEXT, Suffix := Const.CARRIAGE_RETURN);
	{attribute 'OPC.UA.DA' := '0'}
	_refSerialCom : REFERENCE TO SerialCom(Prefix := Const.START_OF_TEXT, Suffix := Const.CARRIAGE_RETURN) := _serialCom;
END_VAR

IF NOT _raiseProperties THEN
	GetStateSignals();
END_IF

// Init device
SUPER^.InitDevice();

IF InitConfigSerialCom AND MppcActivate THEN
	THIS^.Status := TExecutionState.Ready;
ELSE
    THIS^.Status := TExecutionState.Error;	
END_IF

IF THIS^.Status = TExecutionState.Ready THEN
	SUPER^(Conf := _config, SerialCom := _serialCom, RefSerialCom := _refSerialCom);
END_IF

IF SUPER^._initDeviceBase THEN
	IF NOT InitConfigSerialCom THEN
		ConfigureSerialCom();
	ELSIF THIS^.Status = TExecutionState.Ready THEN			
		_refSerialCom(TxBuffer:= HardwareGlobalVariables.TxBufferMppcNarrow, 
					  RxBuffer:= HardwareGlobalVariables.RxBufferMppcNarrow);
		
		// Start Mppc to off 
		IF NOT _initDevice THEN
			InitDevice();
		END_IF				
	END_IF
END_IF

METHOD ConfigureSerialCom
VAR_INPUT
END_VAR

VAR
	Status: INT;
END_VAR
IF _coeAccess.CoeOperation.Ready THEN
	_logger.Information(_message.Reset().Append('Start configuration com serial').ToString());
END_IF;	

_coeAccess.CoeOperation.Start();
_coeAccess(SerialCommunication := _config.SerialCommunication);
	
IF _coeAccess.CoeOperation.Done THEN
	_coeAccess.SetDone();
	
	_Logger.Information(_message.Reset().
							Append('{').Append(TO_STRING(THIS^.Family)).Append('} : ').
							Append(' - Status : ').Append(TO_STRING(_coeAccess.Status)).ToString());
	InitConfigSerialCom := TRUE;
END_IF
 
IF _coeAccess.CoeOperation.Error THEN	
	_coeAccess.SetError(0);
	
	_Logger.Error(_message.Reset().
							Append('{').Append(TO_STRING(THIS^.Family)).Append('} : ').
							Append(' - Status : ').Append(TO_STRING(_coeAccess.Status)).ToString());
	InitConfigSerialCom := TRUE;
END_IF

THIS^.Status := _coeAccess.Status;
State := _coeAccess.Status;
END_METHOD

METHOD FB_init : BOOL
VAR_INPUT
	bInitRetains : BOOL; // if TRUE, the retain variables are initialized (warm start / cold start)
	bInCopyCode : BOOL;  // if TRUE, the instance afterwards gets moved into the copy code (online change)
	Config : C13336MppcConfig;
END_VAR
IF Config.IsEnabled THEN
	_config := Config;
	
	SUPER^._mppcConfig.Name := Config.Name;
	SUPER^._mppcConfig.DeviceID := Config.DeviceID;
	SUPER^._mppcConfig.IsEnabled := Config.IsEnabled;
	SUPER^._mppcConfig.LogLevel := Config.LogLevel;
	
	SUPER^.Name := Config.Name;
	SUPER^.DeviceID := Config.DeviceID;	
	THIS^.Family := DeviceFamily.MPPC;
		
	_Logger.Information(_message.Reset().Append('Init ').
							Append('{').Append(TO_STRING(THIS^.Family)).Append('} - ').
							Append('{').Append(TO_STRING(Config.Name)).Append('}').ToString());																													
END_IF
END_METHOD

METHOD GetStateSignals
VAR_INPUT
END_VAR
VAR
	{attribute 'OPC.UA.DA' := '0'}
	fibersCollector : STRING;
	{attribute 'OPC.UA.DA' := '0'}
	delimeter : STRING := ';';
	{attribute 'OPC.UA.DA' := '0'}
	stateSignal : STRING;
END_VAR

fibersCollector := CONCAT(TO_STRING(EMppcCollector.NARROW), delimeter);

IF NOT InputMppcNarrowStateSignal_1 AND NOT InputMppcNarrowStateSignal_2 THEN
	stateSignal := CONCAT(fibersCollector, TO_STRING(EMppcStateModule.UNRECOVERABLE_ERROR));
ELSIF NOT InputMppcNarrowStateSignal_1 AND InputMppcNarrowStateSignal_2 THEN
	stateSignal := CONCAT(fibersCollector, TO_STRING(EMppcStateModule.AWAITING_COOLING_TEMP_STABLE));
ELSIF InputMppcNarrowStateSignal_1 AND NOT InputMppcNarrowStateSignal_2 THEN
	stateSignal := CONCAT(fibersCollector, TO_STRING(EMppcStateModule.AWAITING_HIGH_VOLTAGE_POWER_SUPPLY_STABLE));
ELSE
	stateSignal := CONCAT(fibersCollector, TO_STRING(EMppcStateModule.MODULE_OPERATING_NORMAL));
END_IF

IF stateSignal <> SUPER^.StateSignalsMsg THEN	
	SUPER^.StateSignalsMsg := stateSignal;
	SUPER^.GetStateSignals();
END_IF
END_METHOD

PROPERTY InitConfigSerialCom : BOOL
GET
InitConfigSerialCom := _initConfigSerialCom;
END_GET
SET
_initConfigSerialCom := InitConfigSerialCom;
END_SET
END_PROPERTY

METHOD InitDevice
VAR_INPUT
END_VAR
VAR	
END_VAR
IF NOT _initDevice THEN		
	IF _pulseGeneratorInit.Q THEN
		_pulseGeneratorInit(IN := FALSE, PT := T#10MS);
			
		CASE _itemInit OF
			0:  _logger.Information(_message.Reset().
								Append(_config.Name).
								Append(' - Start to on').ToString());		
				_itemInit := 1;
				
			1:  _outputVoltageOn := TRUE;			
				_initDevice := TRUE;
				_itemInit := 0;
		END_CASE
	ELSE
		_pulseGeneratorInit(IN := TRUE, PT := T#500MS);	
	END_IF
END_IF
END_METHOD

END_FUNCTION_BLOCK

// ---- PMShared/Hardware/Devices/Shutters/Uniblitz/Ed12dssShutter.TcPOU
{attribute 'OPC.UA.DA' := '1'}
FUNCTION_BLOCK Ed12dssShutter EXTENDS ShutterBase
VAR_INPUT
END_VAR
VAR_OUTPUT
END_VAR
VAR
	{attribute 'OPC.UA.DA' := '0'}
	_config : Ed12dssShutterConfig;		
	{attribute 'OPC.UA.DA' := '0'}
	IoEd12dssShutter : IoEd12dssShutter;
	
	{attribute 'OPC.UA.DA' := '0'}
	_deliverMessages : INT;
	
	ShutterIrisPositionMsg : STRING(255);
	
	{region 'Commands'}
	
	{attribute 'OPC.UA.DA' := '0'}
	_open : BOOL;
	{attribute 'OPC.UA.DA' := '0'}
	_close : BOOL;
	{attribute 'OPC.UA.DA' := '0'}			  		   
	_raiseProperties : BOOL;
			
	{endregion}		

	{attribute 'OPC.UA.DA' := '0'}
	_initDevice : BOOL;	
	
	{attribute 'OPC.UA.DA' := '0'}
	_itemScheduler : INT;	
	{attribute 'OPC.UA.DA' := '0'}
	_pulseGenerator : TON;			
	{attribute 'OPC.UA.DA' := '0'}
	_itemRaisedProperties : INT;

	{attribute 'OPC.UA.DA' := '0'}
	_itemCycling : INT;	
	
	{attribute 'OPC.UA.DA' := '0'}
	message : STRING;
	
	{attribute 'OPC.UA.DA' := '0'}
	_bCycling : BOOL;
		
END_VAR

// Init device
InitDevice();

CASE _deliverMessages OF			
	EFeedbackMsgEd12dss.ShutterIrisPositionMsg :	
		ShutterIrisPositionMsg := message;	
END_CASE
_deliverMessages := 0;
		
// Commands		
ManualOpen(_open);
ManualClose(_close);
Cycling(_bCycling);
RaisePropertiesChanged(_raiseProperties);

IF (NOT _open AND NOT _close AND NOT _raiseProperties) THEN
	MessageScheduler();
END_IF

METHOD PROTECTED Cycling
VAR_INPUT
	Execute : BOOL;
END_VAR
IF Execute THEN			
	IF _pulseGenerator.Q THEN
		_pulseGenerator(IN := FALSE, PT := T#10MS);
		
		CASE _itemCycling OF		
			0: _open := TRUE;
			   _close := FALSE;
				_itemCycling := 1;
				
			1: _open := FALSE;
			   _close := TRUE;
				_itemCycling := 0;
		
		END_CASE	
	ELSE
		_pulseGenerator(IN := TRUE, PT := T#500MS);	
	END_IF									
END_IF
END_METHOD

METHOD FB_init : BOOL
VAR_INPUT
	bInitRetains : BOOL; // if TRUE, the retain variables are initialized (warm start / cold start)
	bInCopyCode : BOOL;  // if TRUE, the instance afterwards gets moved into the copy code (online change)
	Config : Ed12dssShutterConfig;
END_VAR
IF Config.IsEnabled THEN
	_config := Config;
	
	SUPER^._shutterConfig.Name := Config.Name;
	SUPER^._shutterConfig.DeviceID := Config.DeviceID;
	SUPER^._shutterConfig.IsEnabled := Config.IsEnabled;
	SUPER^._shutterConfig.LogLevel := Config.LogLevel;
	
	SUPER^.Name := Config.Name;
	SUPER^.DeviceID := Config.DeviceID;	
	THIS^.Family := DeviceFamily.Shutter;
		
	_Logger.Information(_message.Reset().Append('Init ').
							Append('{').Append(TO_STRING(THIS^.Family)).Append('} - ').
							Append('{').Append(TO_STRING(Config.Name)).Append('}').ToString());																													
END_IF
END_METHOD

METHOD InitDevice
VAR_INPUT
END_VAR
IF NOT _initDevice THEN	
	_logger.Information(_message.Reset().
								Append(_config.Name).
								Append(' - Init device').ToString());
	
	THIS^.SetDone();
	_initDevice := TRUE;	
END_IF
END_METHOD

{attribute 'TcRpcEnable' := '1'}
METHOD PROTECTED ManualClose
VAR_INPUT
	Execute : BOOL;
END_VAR
IF Execute THEN
	_logger.Information(_message.Reset().
								Append(_config.Name).
								Append(' - ManualClose : ').ToString());								
	IoEd12dssShutter.OutputSwitchContactClosure := FALSE;
	_close := FALSE;		
END_IF
END_METHOD

{attribute 'TcRpcEnable' := '1'}
METHOD PROTECTED ManualOpen
VAR_INPUT
	Execute : BOOL;
END_VAR
IF Execute THEN
	_logger.Information(_message.Reset().
								Append(_config.Name).
								Append(' - ManualOpen : ').ToString());		
	IoEd12dssShutter.OutputSwitchContactClosure := TRUE;
	_open := FALSE;		
END_IF
END_METHOD

METHOD MessageScheduler
VAR_INPUT
END_VAR
CASE _itemScheduler OF
		0:  ShutterIrisPosition();		
			_itemScheduler := 0;		
END_CASE
END_METHOD

{attribute 'TcRpcEnable' := '1'}
METHOD RaisePropertiesChanged
VAR_INPUT
	Execute : BOOL;
END_VAR
IF Execute THEN		
	_raiseProperties := TRUE;	
	
	IF _pulseGenerator.Q THEN
		_pulseGenerator(IN := FALSE, PT := T#10MS);
		
		CASE _itemRaisedProperties OF		
			0: ShutterIrisPositionMsg := ' ';		   
				_itemRaisedProperties := 10;
				
			10: 
				_logger.Information(_message.Reset().
								    Append(_config.Name).
								    Append(' - RaisePropertiesChanged').ToString());
				_raiseProperties := FALSE;
				_itemRaisedProperties := 0;
		
		END_CASE
	
	ELSE
		_pulseGenerator(IN := TRUE, PT := T#200MS);	
	END_IF
		
END_IF
END_METHOD

METHOD ShutterIrisPosition 
VAR_INPUT
END_VAR
VAR 
	close : STRING := 'CLOSE';
	open : STRING := 'OPEN';
END_VAR
_deliverMessages := EFeedbackMsgEd12dss.ShutterIrisPositionMsg;

IF IoEd12dssShutter.OutputSwitchContactClosure THEN
	message := open; 	
ELSE
	message := close; 
END_IF
END_METHOD

END_FUNCTION_BLOCK

// ---- PMShared/Hardware/Devices/Shutters/ShutterBase.TcPOU
FUNCTION_BLOCK ABSTRACT ShutterBase EXTENDS TExecution IMPLEMENTS IDevice
VAR_INPUT
END_VAR
VAR_OUTPUT
END_VAR
VAR
	{attribute 'OPC.UA.DA' := '0'}
	_name : STRING;
	{attribute 'OPC.UA.DA' := '0'}
	_deviceID : STRING;				
	{attribute 'OPC.UA.DA' := '0'}	
	_family : DeviceFamily;	
	{attribute 'OPC.UA.DA' := '0'}
	_logger : Logger;
	{attribute 'OPC.UA.DA' := '0'}
	_message : StringBuilder;
	{attribute 'OPC.UA.DA' := '0'}
	_shutterConfig : DeviceConfiguration;	
END_VAR

PROPERTY DeviceID : STRING
GET
DeviceID := _deviceID;
END_GET
SET
_deviceID := DeviceID;
END_SET
END_PROPERTY

PROPERTY Family : DeviceFamily
GET
Family := _family;
END_GET
SET
_family := Family;
END_SET
END_PROPERTY

METHOD PROTECTED ABSTRACT ManualClose
VAR_INPUT
	Execute : BOOL;
END_VAR
END_METHOD

METHOD PROTECTED ABSTRACT ManualOpen
VAR_INPUT
	Execute : BOOL;
END_VAR
END_METHOD

PROPERTY Name : STRING
GET
Name := _name;
END_GET
SET
_name := Name;
END_SET
END_PROPERTY

END_FUNCTION_BLOCK

// ---- PMShared/Hardware/Devices/Shutters/Eopc/Sh10pilShutter.TcPOU
{attribute 'OPC.UA.DA' := '1'}
FUNCTION_BLOCK Sh10pilShutter EXTENDS ShutterBase
VAR_INPUT
END_VAR
VAR_OUTPUT
END_VAR
VAR
	{attribute 'OPC.UA.DA' := '0'}
	_config : Sh10pilShutterConfig;		
	{attribute 'OPC.UA.DA' := '0'}
	IoSh10pilShutter : IoSh10pilShutter;
	
	{attribute 'OPC.UA.DA' := '0'}
	_deliverMessages : INT;
	
	ShutterIrisPositionMsg : STRING(255);
	
	{region 'Commands'}
	
	{attribute 'OPC.UA.DA' := '0'}
	_open : BOOL;
	{attribute 'OPC.UA.DA' := '0'}
	_close : BOOL;
	{attribute 'OPC.UA.DA' := '0'}			  		   
	_raiseProperties : BOOL;
			
	{endregion}		

	{attribute 'OPC.UA.DA' := '0'}
	_initDevice : BOOL;	
	
	{attribute 'OPC.UA.DA' := '0'}
	_itemScheduler : INT;	
	{attribute 'OPC.UA.DA' := '0'}
	_itemOpen : INT;
	{attribute 'OPC.UA.DA' := '0'}
	_itemClose : INT;
	{attribute 'OPC.UA.DA' := '0'}
	_pulseGenerator : TON;	
	{attribute 'OPC.UA.DA' := '0'}
	_pulseOpen : TON;
	{attribute 'OPC.UA.DA' := '0'}
	_pulseClose : TON;
	{attribute 'OPC.UA.DA' := '0'}
	_pulseTimeout : TON;		
	{attribute 'OPC.UA.DA' := '0'}
	_itemRaisedProperties : INT;	
	
	{attribute 'OPC.UA.DA' := '0'}
	message : STRING;
	
END_VAR

// Init device
InitDevice();

CASE _deliverMessages OF			
	EFeedbackMsgSh10pil.ShutterIrisPositionMsg :	
		ShutterIrisPositionMsg := message;	
END_CASE
		
// Commands		
ManualOpen(_open);
ManualClose(_close);
RaisePropertiesChanged(_raiseProperties);

IF (NOT _open AND NOT _close AND NOT _raiseProperties) THEN
	_deliverMessages := 0;
	MessageScheduler();
END_IF

METHOD FB_init : BOOL
VAR_INPUT
	bInitRetains : BOOL; // if TRUE, the retain variables are initialized (warm start / cold start)
	bInCopyCode : BOOL;  // if TRUE, the instance afterwards gets moved into the copy code (online change)
	Config : Sh10pilShutterConfig;
END_VAR
IF Config.IsEnabled THEN
	_config := Config;
	
	SUPER^._shutterConfig.Name := Config.Name;
	SUPER^._shutterConfig.DeviceID := Config.DeviceID;
	SUPER^._shutterConfig.IsEnabled := Config.IsEnabled;
	SUPER^._shutterConfig.LogLevel := Config.LogLevel;
	
	SUPER^.Name := Config.Name;
	SUPER^.DeviceID := Config.DeviceID;	
	THIS^.Family := DeviceFamily.Shutter;
		
	_Logger.Information(_message.Reset().Append('Init ').
							Append('{').Append(TO_STRING(THIS^.Family)).Append('} - ').
							Append('{').Append(TO_STRING(Config.Name)).Append('}').ToString());																													
END_IF
END_METHOD

METHOD InitDevice
VAR_INPUT
END_VAR
IF NOT _initDevice THEN	
	_logger.Information(_message.Reset().
								Append(_config.Name).
								Append(' - Init device').ToString());
	
	THIS^.SetDone();
	_initDevice := TRUE;	
END_IF
END_METHOD

{attribute 'TcRpcEnable' := '1'}
METHOD PROTECTED ManualClose
VAR_INPUT
	Execute : BOOL;
END_VAR
IF Execute THEN	
	_close := TRUE;
	
	CASE _itemClose OF
		0: _logger.Information(_message.Reset().
							Append(_config.Name).
							Append(' - Close').ToString());
							
			_itemClose := 1;
							
		1: //Wait until the shutter is opened 
			IF IoSh10pilShutter.InputMagneticSwitch1 AND NOT IoSh10pilShutter.InputMagneticSwitch2 THEN
				_itemClose := 2;
			ELSE 
				// Raised timer 
				IF _pulseTimeout.Q THEN
					_pulseTimeout(IN := FALSE);
					
					_itemClose := 2;
				ELSE
					_pulseTimeout(IN := TRUE, PT := T#100MS);	
				END_IF	
			END_IF 
			
		2: IF _pulseOpen.Q THEN
				_pulseOpen(IN := FALSE);
				
				IoSh10pilShutter.OutputSwitchContactClosure := FALSE;
				_close := FALSE;
				_itemClose := 0;
			ELSE
				_pulseOpen(IN := TRUE, PT := T#10MS);	
			END_IF		
							
	END_CASE

END_IF
END_METHOD

{attribute 'TcRpcEnable' := '1'}
METHOD PROTECTED ManualOpen
VAR_INPUT
	Execute : BOOL;
END_VAR
IF Execute THEN
	_open := TRUE;
	
	CASE _itemOpen OF
		0: _logger.Information(_message.Reset().
							Append(_config.Name).
							Append(' - Open').ToString());
							
			_itemOpen := 1;
							
		1: //Wait until the shutter is closed 
			IF NOT IoSh10pilShutter.InputMagneticSwitch1 AND IoSh10pilShutter.InputMagneticSwitch2 THEN
				_itemOpen := 2;
			ELSE
				// Raised timer 
				IF _pulseTimeout.Q THEN
					_pulseTimeout(IN := FALSE);
					
					_itemOpen := 2;
				ELSE
					_pulseTimeout(IN := TRUE, PT := T#100MS);	
				END_IF	
			END_IF 
			
		2: IF _pulseOpen.Q THEN
				_pulseOpen(IN := FALSE);
				
				IoSh10pilShutter.OutputSwitchContactClosure := TRUE;
				_open := FALSE;
				_itemOpen := 0;
			ELSE
				_pulseOpen(IN := TRUE, PT := T#400MS);	
			END_IF		
							
	END_CASE
	
END_IF
END_METHOD

METHOD MessageScheduler
VAR_INPUT
END_VAR
IF _pulseGenerator.Q THEN
	_pulseGenerator(IN := FALSE, PT := T#10MS);
	
	ShutterIrisPosition();
ELSE
	_pulseGenerator(IN := TRUE, PT := T#100MS);		
END_IF
END_METHOD

{attribute 'TcRpcEnable' := '1'}
METHOD RaisePropertiesChanged
VAR_INPUT
	Execute : BOOL;
END_VAR
IF Execute THEN		
	_raiseProperties := TRUE;	
	
	IF _pulseGenerator.Q THEN
		_pulseGenerator(IN := FALSE, PT := T#10MS);
		
		CASE _itemRaisedProperties OF		
			0: ShutterIrisPositionMsg := ' ';
				_itemRaisedProperties := 1;
			
			1: ShutterIrisPosition();		   
				_itemRaisedProperties := 10;
				
			10: 
				_logger.Information(_message.Reset().
								    Append(_config.Name).
								    Append(' - RaisePropertiesChanged').ToString());
				_raiseProperties := FALSE;
				_itemRaisedProperties := 0;
		
		END_CASE
	
	ELSE
		_pulseGenerator(IN := TRUE, PT := T#200MS);	
	END_IF
		
END_IF
END_METHOD

METHOD ShutterIrisPosition 
VAR_INPUT
END_VAR
VAR 
	close : STRING := 'CLOSE';
	open : STRING := 'OPEN';
	error : STRING := 'ERROR';
END_VAR
_deliverMessages := EFeedbackMsgEd12dss.ShutterIrisPositionMsg;

IF IoSh10pilShutter.InputMagneticSwitch1 AND NOT IoSh10pilShutter.InputMagneticSwitch2 THEN
	message := open; 		
ELSIF NOT IoSh10pilShutter.InputMagneticSwitch1 AND IoSh10pilShutter.InputMagneticSwitch2 THEN
	message := close; 
ELSIF IoSh10pilShutter.InputMagneticSwitch1 AND IoSh10pilShutter.InputMagneticSwitch2 THEN
	message := error; 
END_IF
END_METHOD

END_FUNCTION_BLOCK

// ---- PMShared/Hardware/Devices/FastAttenuation/Parallax/Std900FastAttenuation.TcPOU
FUNCTION_BLOCK Std900FastAttenuation EXTENDS FastAttenuationBase
VAR_INPUT
END_VAR
VAR_OUTPUT
END_VAR
VAR
	{attribute 'OPC.UA.DA' := '0'}
	_config : Std900FastAttenuationConfig;
	{attribute 'OPC.UA.DA' := '0'}
	IoStd900 : IoStd900;
	
	{attribute 'OPC.UA.DA' := '0'}
	_deliverMessages : INT;
	
	PositionMsg : STRING(255);
	
	{region 'Commands'}	
		 
	{attribute 'OPC.UA.DA' := '0'}
	_moveAbsPosition	 : BOOL;
		 
	{endregion}
		 
	{attribute 'OPC.UA.DA' := '0'}
	_initDevice : BOOL;	
		
	{attribute 'OPC.UA.DA' := '0'}
	_pos : UINT;
	{attribute 'OPC.UA.DA' := '0'}
	_itemScheduler : INT;
	{attribute 'OPC.UA.DA' := '0'}
	_pulseGenerator : TON;		
END_VAR

// Init device
InitDevice(); 	
			  
// Deliver messages
CASE _deliverMessages OF	
		EFeedbackMsgStd900.PositionMsg :
		PositionMsg := REAL_TO_STRING(GetPosition());			
END_CASE
	
_deliverMessages := 0;

// Commands
MoveAbsPosition(_moveAbsPosition, _pos); 

IF NOT _moveAbsPosition THEN
	MessageScheduler();
END_IF

METHOD FB_init : BOOL
VAR_INPUT
	bInitRetains : BOOL; // if TRUE, the retain variables are initialized (warm start / cold start)
	bInCopyCode : BOOL;  // if TRUE, the instance afterwards gets moved into the copy code (online change)
	Config : Std900FastAttenuationConfig;
END_VAR
IF Config.IsEnabled THEN
	_config := Config;
	
	SUPER^._fastAttenuationConfig.Name := Config.Name;
	SUPER^._fastAttenuationConfig.DeviceID := Config.DeviceID;
	SUPER^._fastAttenuationConfig.IsEnabled := Config.IsEnabled;
	SUPER^._fastAttenuationConfig.LogLevel := Config.LogLevel;
	
	SUPER^.Name := Config.Name;
	SUPER^.DeviceID := Config.DeviceID;	
	THIS^.Family := DeviceFamily.FastAttenuation;
	
	_Logger.Information(_message.Reset().Append('Init ').
							Append('{').Append(TO_STRING(THIS^.Family)).Append('} - ').
							Append('{').Append(TO_STRING(Config.Name)).Append('}').ToString());																													
END_IF
END_METHOD

METHOD GetPosition : REAL
VAR_INPUT
END_VAR
_deliverMessages := EFeedbackMsgStd900.PositionMsg;

GetPosition := ((IoStd900.OutputPwm - Const.STD900_LOW_LIMIT) * Const.STD900_MAX_ANGLE) / (Const.STD900_HIGHT_LIMIT - Const.STD900_LOW_LIMIT);
END_METHOD

METHOD InitDevice : BOOL
VAR_INPUT
END_VAR
IF NOT _initDevice THEN	
	_logger.Information(_message.Reset().
								Append(_config.Name).
								Append(' - Init device').ToString());
							
	THIS^.Status := TExecutionState.Ready;
	
	IF IoStd900.OutputPwm = 0 THEN
		MoveAbsPosition(TRUE, 0);
	END_IF
	GetPosition();
	
	_initDevice := TRUE;	
END_IF
END_METHOD

METHOD MessageScheduler
VAR_INPUT
END_VAR
IF _pulseGenerator.Q THEN
	_pulseGenerator(IN := FALSE, PT := T#10MS);
		
	CASE _itemScheduler OF	
		0:	GetPosition();
			_itemScheduler := 1;	
		
		1 : 
			_itemScheduler := 0;											
	END_CASE
ELSE
	_pulseGenerator(IN := TRUE, PT := T#100MS);	
END_IF
END_METHOD

{attribute 'TcRpcEnable' := '1'}
METHOD PROTECTED MoveAbsPosition 
VAR_INPUT
	Execute : BOOL;
	AnglePosition : LREAL;
END_VAR
VAR
	pulseLength : LREAL;
END_VAR
IF Execute THEN
	_logger.Information(_message.Reset().
								Append(_config.Name).
								Append(' - Move absolute position : ').Append(TO_STRING(AnglePosition)).ToString());
	
	_moveAbsPosition := FALSE;
	
	IF AnglePosition >= Const.STD900_MIN_ANGLE AND AnglePosition <= Const.STD900_MAX_ANGLE THEN
		
		IF AnglePosition = Const.STD900_MIN_ANGLE THEN
			pulseLength := Const.STD900_LOW_LIMIT;		
		ELSE
			pulseLength := (Const.STD900_HIGHT_LIMIT - Const.STD900_LOW_LIMIT) / (Const.STD900_MAX_ANGLE / AnglePosition) + Const.STD900_LOW_LIMIT;
		END_IF
		
		_logger.Information(_message.Reset().
								Append('Pulse length : ').Append(TO_STRING(pulseLength)).
								Append(' µs').ToString());
		
		IoStd900.OutputPwm := LREAL_TO_UINT(pulseLength);
		IoStd900.OutputPeriodPwm := Const.STD900_INTERVAL + LREAL_TO_UINT(pulseLength);
	
	END_IF
	
	_itemScheduler := 0;
END_IF
END_METHOD

{attribute 'TcRpcEnable' := '1'}
METHOD RaisePropertiesChanged
VAR_INPUT
	Execute : BOOL;
END_VAR
IF Execute THEN
	PositionMsg := ' ';
END_IF
END_METHOD

END_FUNCTION_BLOCK

// ---- PMShared/Hardware/Devices/FastAttenuation/FastAttenuationBase.TcPOU
FUNCTION_BLOCK ABSTRACT FastAttenuationBase EXTENDS TExecution IMPLEMENTS IDevice
VAR_INPUT
END_VAR
VAR_OUTPUT
END_VAR
VAR
	{attribute 'OPC.UA.DA' := '0'}
	_name : STRING;
	{attribute 'OPC.UA.DA' := '0'}
	_deviceID : STRING;					
	{attribute 'OPC.UA.DA' := '0'}
	_family : DeviceFamily;				
	{attribute 'OPC.UA.DA' := '0'}
	_logger : Logger;
	{attribute 'OPC.UA.DA' := '0'}
	_message : StringBuilder;	
	{attribute 'OPC.UA.DA' := '0'}
	_fastAttenuationConfig : DeviceConfiguration;
END_VAR

PROPERTY DeviceID : STRING
GET
DeviceID := _deviceID;
END_GET
SET
_deviceID := DeviceID;
END_SET
END_PROPERTY

PROPERTY Family : DeviceFamily
GET
Family := _family;
END_GET
SET
_family := Family;
END_SET
END_PROPERTY

METHOD PROTECTED ABSTRACT MoveAbsPosition
VAR_INPUT
	Execute : BOOL;
	AnglePosition : LREAL;
END_VAR
END_METHOD

PROPERTY Name : STRING
GET
Name := _name;
END_GET
SET
_name := Name;
END_SET
END_PROPERTY

END_FUNCTION_BLOCK

// ---- Service/PMs/Lightspeed/Communication/RS232/LsBkgrdLsSerialCom.TcPOU
PROGRAM LsBkgrdLsSerialCom
VAR_INPUT
	Config : LightspeedConfig;
END_VAR
VAR
END_VAR

// AttenuationFilterConfigs
IF Config.AttenuationFilterConfigs.FW212CAttenuationFilterConfig.IsEnabled OR 
   Config.AttenuationFilterConfigs.ELL14kAttenuationFilterConfig.IsEnabled OR
   Config.AttenuationFilterConfigs.ELL9AttenuationFilterConfig.IsEnabled THEN
	BkgrdSerialAttenuation();	
END_IF

// SliderAttenuationFilterConfigs
IF Config.SliderAttenuationFilterConfigs.ELL6SliderFilterConfig.IsEnabled THEN
	BkgrdSerialSliderAttenuation();	
END_IF

// RotatingSwitchConfigs
IF Config.RotatingSwitchConfigs.ELL18RotatingSwitchConfig.IsEnabled THEN
	BkgrdSerialRotatingSwitch();	
END_IF

// PolarisationFilterConfigs
IF Config.PolarisationFilterConfigs.FW212CPolarisationFilterConfig.IsEnabled OR 
   Config.PolarisationFilterConfigs.ELL14KPolarisationFilterConfig.IsEnabled THEN
	BkgrdSerialPolarisation();		
END_IF

// LaserConfigs
IF Config.LaserConfigs.SMD12LaserConfig.IsEnabled OR 
	Config.LaserConfigs.Sapphire488LaserConfig.IsEnabled THEN
	BkgrdSerialLaser();
END_IF

// FiberSwitchConfigs
IF Config.FiberSwitchConfigs.EOLFiberSwitchConfig.IsEnabled THEN
	BkgrdSerialFiberSwitch();
END_IF

// OpticalPowermeterConfigs
IF Config.OpticalPowermeterConfigs.PM101OpticalPowermeterConfigHs.IsEnabled THEN
	BkgrdSerialOpticalPowermeterHs();	
END_IF
IF Config.OpticalPowermeterConfigs.PM101OpticalPowermeterConfigHt.IsEnabled THEN
	BkgrdSerialOpticalPowermeterHt();	
END_IF

// MppcConfigs
IF Config.MppcConfigs.C13336MppcConfigWide.IsEnabled THEN
	BkgrdSerialMppcWide();
END_IF
IF Config.MppcConfigs.C13336MppcConfigNarrow.IsEnabled THEN
	BkgrdSerialMppcNarrow();
END_IF

END_PROGRAM

// ---- PMShared/Hardware/Devices/AttenuationFilters/Configs/SerialCommunication/BkgrdSerialAttenuation.TcPOU
PROGRAM BkgrdSerialAttenuation
VAR
	(* background communication with the EL6002 terminal *)
	serialLineCtrl		: SerialLineControl;
	serialLineCtrlError	: BOOL;
	serialLineCtrlErrorID : ComError_t;
	(* 	I/O variables for a EL6002 terminal*)
	stInAttenuation  AT %I*	: EL6inData22B;	
	stOutAttenuation AT %Q*	: EL6outData22B;
END_VAR

(*
The SerialLineControl function block is supposed to be called in every PLC cycle.
It communicates with the serial line hardware device and transmits or receives data.
The SerialLineControl can be called in the standard task (e.g.for PcCOM port usage) 
or in a separate fast task (e.g.for terminal usage) as well.
A fast separate task will be necessary at high baud rates or with KL6001 terminals 
which have a small process image (3 or 5 data bytes only)
*)

(* background communication with the EL6002 terminal *)
serialLineCtrl(
	Mode:= SERIALLINEMODE_EL6_22B, 
	pComIn:= ADR(stInAttenuation), 
	pComOut:= ADR(stOutAttenuation), 
	SizeComIn:= SIZEOF(stInAttenuation), 
	TxBuffer:= HardwareGlobalVariables.TxBufferAttenuation, 
	RxBuffer:= HardwareGlobalVariables.RxBufferAttenuation
);

IF serialLineCtrl.Error THEN
	serialLineCtrlError := TRUE;
	serialLineCtrlErrorID := serialLineCtrl.ErrorID;
END_IF

END_PROGRAM

// ---- PMShared/Hardware/Devices/AttenuationFilters/Configs/SerialCommunication/BkgrdSerialSliderAttenuation.TcPOU
PROGRAM BkgrdSerialSliderAttenuation
VAR
	(* background communication with the EL6002 terminal *)
	serialLineCtrl		: SerialLineControl;
	serialLineCtrlError	: BOOL;
	serialLineCtrlErrorID : ComError_t;
	(* 	I/O variables for a EL6002 terminal*)
	stInSliderAttenuation  AT %I*	: EL6inData22B;	
	stOutSliderAttenuation AT %Q*	: EL6outData22B;
END_VAR

(*
The SerialLineControl function block is supposed to be called in every PLC cycle.
It communicates with the serial line hardware device and transmits or receives data.
The SerialLineControl can be called in the standard task (e.g.for PcCOM port usage) 
or in a separate fast task (e.g.for terminal usage) as well.
A fast separate task will be necessary at high baud rates or with KL6001 terminals 
which have a small process image (3 or 5 data bytes only)
*)

(* background communication with the EL6002 terminal *)
serialLineCtrl(
	Mode:= SERIALLINEMODE_EL6_22B, 
	pComIn:= ADR(stInSliderAttenuation), 
	pComOut:= ADR(stOutSliderAttenuation), 
	SizeComIn:= SIZEOF(stInSliderAttenuation), 
	TxBuffer:= HardwareGlobalVariables.TxBufferSliderAttenuation, 
	RxBuffer:= HardwareGlobalVariables.RxBufferSliderAttenuation
);

IF serialLineCtrl.Error THEN
	serialLineCtrlError := TRUE;
	serialLineCtrlErrorID := serialLineCtrl.ErrorID;
END_IF

END_PROGRAM

// ---- PMShared/Hardware/Devices/AttenuationFilters/Configs/SerialCommunication/BkgrdSerialRotatingSwitch.TcPOU
PROGRAM BkgrdSerialRotatingSwitch
VAR
	(* background communication with the EL6002 terminal *)
	serialLineCtrl		: SerialLineControl;
	serialLineCtrlError	: BOOL;
	serialLineCtrlErrorID : ComError_t;
	(* 	I/O variables for a EL6002 terminal*)
	stInRotatingSwitch  AT %I*	: EL6inData22B;	
	stOutRotatingSwitch AT %Q*	: EL6outData22B;
END_VAR

(*
The SerialLineControl function block is supposed to be called in every PLC cycle.
It communicates with the serial line hardware device and transmits or receives data.
The SerialLineControl can be called in the standard task (e.g.for PcCOM port usage) 
or in a separate fast task (e.g.for terminal usage) as well.
A fast separate task will be necessary at high baud rates or with KL6001 terminals 
which have a small process image (3 or 5 data bytes only)
*)

(* background communication with the EL6002 terminal *)
serialLineCtrl(
	Mode:= SERIALLINEMODE_EL6_22B, 
	pComIn:= ADR(stInRotatingSwitch), 
	pComOut:= ADR(stOutRotatingSwitch), 
	SizeComIn:= SIZEOF(stInRotatingSwitch), 
	TxBuffer:= HardwareGlobalVariables.TxBufferRotatingSwitch, 
	RxBuffer:= HardwareGlobalVariables.RxBufferRotatingSwitch
);

IF serialLineCtrl.Error THEN
	serialLineCtrlError := TRUE;
	serialLineCtrlErrorID := serialLineCtrl.ErrorID;
END_IF

END_PROGRAM

// ---- PMShared/Hardware/Devices/PolarisationFilters/Configs/SerialCommunication/BkgrdSerialPolarisation.TcPOU
PROGRAM BkgrdSerialPolarisation
VAR
	(* background communication with the EL6002 terminal *)
	serialLineCtrl		: SerialLineControl;
	serialLineCtrlError	: BOOL;
	serialLineCtrlErrorID : ComError_t;
	(* 	I/O variables for a EL6002 terminal*)
	stInPolarisation  AT %I* : EL6inData22B;	
	stOutPolarisation AT %Q* : EL6outData22B;
END_VAR

(*
The SerialLineControl function block is supposed to be called in every PLC cycle.
It communicates with the serial line hardware device and transmits or receives data.
The SerialLineControl can be called in the standard task (e.g.for PcCOM port usage) 
or in a separate fast task (e.g.for terminal usage) as well.
A fast separate task will be necessary at high baud rates or with KL6001 terminals 
which have a small process image (3 or 5 data bytes only)
*)

(* background communication with the EL6002 terminal *)
serialLineCtrl(
	Mode:= SERIALLINEMODE_EL6_22B, 
	pComIn:= ADR(stInPolarisation), 
	pComOut:= ADR(stOutPolarisation), 
	SizeComIn:= SIZEOF(stInPolarisation),
	TxBuffer:= HardwareGlobalVariables.TxBufferPolarisation, 
	RxBuffer:= HardwareGlobalVariables.RxBufferPolarisation
);

IF serialLineCtrl.Error THEN
	serialLineCtrlError := TRUE;
	serialLineCtrlErrorID := serialLineCtrl.ErrorID;
END_IF

END_PROGRAM

// ---- PMShared/Hardware/Devices/Lasers/Configs/SerialCommunication/BkgrdSerialLaser.TcPOU
PROGRAM BkgrdSerialLaser
VAR
	(* background communication with the EL6002 terminal *)
	serialLineCtrl		: SerialLineControl;
	serialLineCtrlError	: BOOL;
	serialLineCtrlErrorID : ComError_t;
	(* 	I/O variables for a EL6002 terminal*)
	stInLaser  AT %I* : EL6inData22B;	
	stOutLaser AT %Q* : EL6outData22B;
END_VAR

(*
The SerialLineControl function block is supposed to be called in every PLC cycle.
It communicates with the serial line hardware device and transmits or receives data.
The SerialLineControl can be called in the standard task (e.g.for PcCOM port usage) 
or in a separate fast task (e.g.for terminal usage) as well.
A fast separate task will be necessary at high baud rates or with KL6001 terminals 
which have a small process image (3 or 5 data bytes only)
*)

(* background communication with the EL6002 terminal *)
serialLineCtrl(
	Mode:= SERIALLINEMODE_EL6_22B, 
	pComIn:= ADR(stInLaser), 
	pComOut:= ADR(stOutLaser), 
	SizeComIn:= SIZEOF(stInLaser), 
	TxBuffer:= HardwareGlobalVariables.TxBufferLaser, 
	RxBuffer:= HardwareGlobalVariables.RxBufferLaser
);

IF serialLineCtrl.Error THEN
	serialLineCtrlError := TRUE;
	serialLineCtrlErrorID := serialLineCtrl.ErrorID;
END_IF

END_PROGRAM

// ---- PMShared/Hardware/Devices/FiberSwitch/Configs/SerialCommunication/BkgrdSerialFiberSwitch.TcPOU
PROGRAM BkgrdSerialFiberSwitch
VAR
	(* background communication with the EL6002 terminal *)
	serialLineCtrl		: SerialLineControl;
	serialLineCtrlError	: BOOL;
	serialLineCtrlErrorID : ComError_t;
	(* 	I/O variables for a EL6002 terminal*)
	stInFiberSwitch  AT %I*	: EL6inData22B;	
	stOutFiberSwitch AT %Q*	: EL6outData22B;
END_VAR

(*
The SerialLineControl function block is supposed to be called in every PLC cycle.
It communicates with the serial line hardware device and transmits or receives data.
The SerialLineControl can be called in the standard task (e.g.for PcCOM port usage) 
or in a separate fast task (e.g.for terminal usage) as well.
A fast separate task will be necessary at high baud rates or with KL6001 terminals 
which have a small process image (3 or 5 data bytes only)
*)

(* background communication with the EL6002 terminal *)
serialLineCtrl(
	Mode:= SERIALLINEMODE_EL6_22B, 
	pComIn:= ADR(stInFiberSwitch), 
	pComOut:= ADR(stOutFiberSwitch), 
	SizeComIn:= SIZEOF(stInFiberSwitch), 
	TxBuffer:= HardwareGlobalVariables.TxBufferFiberSwitch, 
	RxBuffer:= HardwareGlobalVariables.RxBufferFiberSwitch
);

IF serialLineCtrl.Error THEN
	serialLineCtrlError := TRUE;
	serialLineCtrlErrorID := serialLineCtrl.ErrorID;
END_IF

END_PROGRAM

// ---- PMShared/Hardware/Devices/OpticalPowermeters/Configs/SerialCommunication/BkgrdSerialOpticalPowermeterHs.TcPOU
PROGRAM BkgrdSerialOpticalPowermeterHs
VAR
	(* background communication with the EL6002 terminal *)
	serialLineCtrl		: SerialLineControl;
	serialLineCtrlError	: BOOL;
	serialLineCtrlErrorID : ComError_t;
	(* 	I/O variables for a EL6002 terminal*)
	stInThorlabsOpticalPowermeterHs  AT %I* : EL6inData22B;	
	stOutThorlabsOpticalPowermeterHs AT %Q* : EL6outData22B;
END_VAR

(*
The SerialLineControl function block is supposed to be called in every PLC cycle.
It communicates with the serial line hardware device and transmits or receives data.
The SerialLineControl can be called in the standard task (e.g.for PcCOM port usage) 
or in a separate fast task (e.g.for terminal usage) as well.
A fast separate task will be necessary at high baud rates or with KL6001 terminals 
which have a small process image (3 or 5 data bytes only)
*)

(* background communication with the EL6002 terminal *)
serialLineCtrl(
	Mode:= SERIALLINEMODE_EL6_22B, 
	pComIn:= ADR(stInThorlabsOpticalPowermeterHs), 
	pComOut:= ADR(stOutThorlabsOpticalPowermeterHs), 
	SizeComIn:= SIZEOF(stInThorlabsOpticalPowermeterHs), 
	TxBuffer:= HardwareGlobalVariables.TxBufferOpticalPowermeterHs, 
	RxBuffer:= HardwareGlobalVariables.RxBufferOpticalPowermeterHs
);

IF serialLineCtrl.Error THEN
	serialLineCtrlError := TRUE;
	serialLineCtrlErrorID := serialLineCtrl.ErrorID;
END_IF

END_PROGRAM

// ---- PMShared/Hardware/Devices/OpticalPowermeters/Configs/SerialCommunication/BkgrdSerialOpticalPowermeterHt.TcPOU
PROGRAM BkgrdSerialOpticalPowermeterHt
VAR
	(* background communication with the EL6002 terminal *)
	serialLineCtrl		: SerialLineControl;
	serialLineCtrlError	: BOOL;
	serialLineCtrlErrorID : ComError_t;
	(* 	I/O variables for a EL6002 terminal*)
	stInThorlabsOpticalPowermeterHt  AT %I* : EL6inData22B;	
	stOutThorlabsOpticalPowermeterHt AT %Q* : EL6outData22B;
END_VAR

(*
The SerialLineControl function block is supposed to be called in every PLC cycle.
It communicates with the serial line hardware device and transmits or receives data.
The SerialLineControl can be called in the standard task (e.g.for PcCOM port usage) 
or in a separate fast task (e.g.for terminal usage) as well.
A fast separate task will be necessary at high baud rates or with KL6001 terminals 
which have a small process image (3 or 5 data bytes only)
*)

(* background communication with the EL6002 terminal *)
serialLineCtrl(
	Mode:= SERIALLINEMODE_EL6_22B, 
	pComIn:= ADR(stInThorlabsOpticalPowermeterHt), 
	pComOut:= ADR(stOutThorlabsOpticalPowermeterHt), 
	SizeComIn:= SIZEOF(stInThorlabsOpticalPowermeterHt), 
	TxBuffer:= HardwareGlobalVariables.TxBufferOpticalPowermeterHt, 
	RxBuffer:= HardwareGlobalVariables.RxBufferOpticalPowermeterHt
	
);

IF serialLineCtrl.Error THEN
	serialLineCtrlError := TRUE;
	serialLineCtrlErrorID := serialLineCtrl.ErrorID;
END_IF

END_PROGRAM

// ---- PMShared/Hardware/Devices/MPPCs/Configs/SerialCommunication/BkgrdSerialMppcWide.TcPOU
PROGRAM BkgrdSerialMppcWide
VAR
	(* background communication with the EL6002 terminal *)
	serialLineCtrl		: SerialLineControl;
	serialLineCtrlError	: BOOL;
	serialLineCtrlErrorID : ComError_t;
	(* 	I/O variables for a EL6002 terminal*)
	stInMppcWide  AT %I*	: EL6inData22B;	
	stOutMppcWide AT %Q*	: EL6outData22B;
END_VAR

(*
The SerialLineControl function block is supposed to be called in every PLC cycle.
It communicates with the serial line hardware device and transmits or receives data.
The SerialLineControl can be called in the standard task (e.g.for PcCOM port usage) 
or in a separate fast task (e.g.for terminal usage) as well.
A fast separate task will be necessary at high baud rates or with KL6001 terminals 
which have a small process image (3 or 5 data bytes only)
*)

(* background communication with the EL6002 terminal *)
serialLineCtrl(
	Mode:= SERIALLINEMODE_EL6_22B, 
	pComIn:= ADR(stInMppcWide), 
	pComOut:= ADR(stOutMppcWide), 
	SizeComIn:= SIZEOF(stInMppcWide), 
	TxBuffer:= HardwareGlobalVariables.TxBufferMppcWide, 
	RxBuffer:= HardwareGlobalVariables.RxBufferMppcWide
);

IF serialLineCtrl.Error THEN
	serialLineCtrlError := TRUE;
	serialLineCtrlErrorID := serialLineCtrl.ErrorID;
END_IF

END_PROGRAM

// ---- PMShared/Hardware/Devices/MPPCs/Configs/SerialCommunication/BkgrdSerialMppcNarrow.TcPOU
PROGRAM BkgrdSerialMppcNarrow
VAR
	(* background communication with the EL6002 terminal *)
	serialLineCtrl		: SerialLineControl;
	serialLineCtrlError	: BOOL;
	serialLineCtrlErrorID : ComError_t;
	(* 	I/O variables for a EL6002 terminal*)
	stInMppcNarrow  AT %I*	: EL6inData22B;	
	stOutMppcNarrow AT %Q*	: EL6outData22B;
END_VAR

(*
The SerialLineControl function block is supposed to be called in every PLC cycle.
It communicates with the serial line hardware device and transmits or receives data.
The SerialLineControl can be called in the standard task (e.g.for PcCOM port usage) 
or in a separate fast task (e.g.for terminal usage) as well.
A fast separate task will be necessary at high baud rates or with KL6001 terminals 
which have a small process image (3 or 5 data bytes only)
*)

(* background communication with the EL6002 terminal *)
serialLineCtrl(
	Mode:= SERIALLINEMODE_EL6_22B, 
	pComIn:= ADR(stInMppcNarrow), 
	pComOut:= ADR(stOutMppcNarrow), 
	SizeComIn:= SIZEOF(stInMppcNarrow), 
	TxBuffer:= HardwareGlobalVariables.TxBufferMppcNarrow, 
	RxBuffer:= HardwareGlobalVariables.RxBufferMppcNarrow
);

IF serialLineCtrl.Error THEN
	serialLineCtrlError := TRUE;
	serialLineCtrlErrorID := serialLineCtrl.ErrorID;
END_IF

END_PROGRAM

// ---- Service/PMs/Psd/Psd.TcPOU
FUNCTION_BLOCK Psd EXTENDS PlcModule
VAR_INPUT	
	Safety : Safety;
	
	{attribute 'OPC.UA.DA' := '0'}
	PsdConfig : PsdConfig;
	
	(* Axes *)
	IoStageAxis : IoStageAxis(Config := PsdConfig.AxesConfigs.IoStageAxisConfig);
	
	(* Chamber *)
	Chamber : PsdChamber(Config := PsdConfig.ChamberConfigs.PsdChamberConfig);
	
	(* Chuck *)
	Chuck : PsdChuck(Config := PsdConfig.ChuckConfigs.PsdChuckConfig);
	
	(* Ffu *)
	Ffu : Astrofan612Ffu(Config := PsdConfig.FfuConfigs.Astrofan612FfuConfig);
	
	(* Screen *)
	DM430GNScreenFS : DM430GNScreenFS(Config := PsdConfig.ScreenConfigs.DM430GNScreenConfigFS);
	DM430GNScreenBS : DM430GNScreenBS(Config := PsdConfig.ScreenConfigs.DM430GNScreenConfigBS);
	
	(* RFid *)
	Rfid : BisL405Rfid(Config := PsdConfig.RfidConfigs.BisL405RfidConfig);		
	
END_VAR
VAR_OUTPUT
END_VAR
VAR
END_VAR

SUPER^();

IF PsdConfig.SafetyIsEnabled THEN
	Safety();
END_IF

IF PsdConfig.AxesConfigs.IoStageAxisConfig.IsEnabled THEN
	IoStageAxis();	
END_IF

IF PsdConfig.ChamberConfigs.PsdChamberConfig.IsEnabled THEN
	Chamber();		
END_IF

IF PsdConfig.ChuckConfigs.PsdChuckConfig.IsEnabled THEN
	Chuck();		
END_IF

IF PsdConfig.FfuConfigs.Astrofan612FfuConfig.IsEnabled THEN
	Ffu();	
END_IF
	
// Screens
IF PsdConfig.ScreenConfigs.DM430GNScreenConfigFS.IsEnabled THEN
	DM430GNScreenFS();
	IF DM430GNScreenFS.InitConfigSerialCom THEN
		;
	END_IF
END_IF

IF PsdConfig.ScreenConfigs.DM430GNScreenConfigBS.IsEnabled THEN
	DM430GNScreenBS();
	IF DM430GNScreenBS.InitConfigSerialCom THEN
		;
	END_IF
END_IF

IF PsdConfig.RfidConfigs.BisL405RfidConfig.IsEnabled THEN
	Rfid();	
END_IF


IF IoStageAxis.GetPosition() = EStagePosition.Loading THEN
	Chamber.StageIsInLoadingPosition := TRUE;	
ELSE
	Chamber.StageIsInLoadingPosition := FALSE;
END_IF

METHOD FB_init : BOOL
VAR_INPUT
	bInitRetains : BOOL; // if TRUE, the retain variables are initialized (warm start / cold start)
	bInCopyCode : BOOL;  // if TRUE, the instance afterwards gets moved into the copy code (online change)
	Config : PsdConfig;
END_VAR
PsdConfig := Config;
PsdBkgrdSerialCom(Config := PsdConfig);

IF Config.IsEnabled THEN
	_logger.Information('Psd devices initialization starting...');
END_IF

// Axis
IF Config.AxesConfigs.IoStageAxisConfig.IsEnabled THEN
	IoStageAxis.FB_init(FALSE, FALSE, Config := Config.AxesConfigs.IoStageAxisConfig);	
END_IF

// Chamber
IF Config.ChamberConfigs.PsdChamberConfig.IsEnabled THEN
	Chamber.FB_init(FALSE, FALSE, Config := Config.ChamberConfigs.PsdChamberConfig);	
END_IF

// Chuck
IF Config.ChuckConfigs.PsdChuckConfig.IsEnabled THEN
	Chuck.FB_init(FALSE, FALSE, Config := Config.ChuckConfigs.PsdChuckConfig);	
END_IF

// FFU
IF Config.FfuConfigs.Astrofan612FfuConfig.IsEnabled THEN
	Ffu.FB_init(FALSE, FALSE, Config := Config.FfuConfigs.Astrofan612FfuConfig);	
END_IF

// Screens
IF Config.ScreenConfigs.DM430GNScreenConfigFS.IsEnabled THEN
	DM430GNScreenFS.FB_init(FALSE, FALSE, Config := Config.ScreenConfigs.DM430GNScreenConfigFS);	
END_IF
IF Config.ScreenConfigs.DM430GNScreenConfigBS.IsEnabled THEN
	DM430GNScreenBS.FB_init(FALSE, FALSE, Config := Config.ScreenConfigs.DM430GNScreenConfigBS);	
END_IF

// RFid
IF Config.RfidConfigs.BisL405RfidConfig.IsEnabled THEN
	Rfid.FB_init(FALSE, FALSE, Config := Config.RfidConfigs.BisL405RfidConfig);	
END_IF

IF Config.IsEnabled THEN
	_logger.Information('Psd devices initialization ended...');
END_IF
END_METHOD

END_FUNCTION_BLOCK

// ---- PMShared/Hardware/Devices/Safety/Safety.TcPOU
FUNCTION_BLOCK Safety
VAR_INPUT	
END_VAR
VAR_OUTPUT
END_VAR
VAR
	{attribute 'OPC.UA.DA' := '0'}
	_message : StringBuilder;
	{attribute 'OPC.UA.DA' := '0'}
	_logger : Logger;
	
	{attribute 'OPC.UA.DA' := '0'}
	_execStartSafety : BOOL := TRUE;	
	{attribute 'OPC.UA.DA' := '0'}
	_execErrAcq : BOOL; 

	{attribute 'OPC.UA.DA' := '0'}
	GroupComErr AT %I* : BOOL;
	{attribute 'OPC.UA.DA' := '0'}
	GroupComStartup AT %I* : BOOL;
	{attribute 'OPC.UA.DA' := '0'}
	GroupFBDeactivate AT %I* : BOOL;
	{attribute 'OPC.UA.DA' := '0'}
	GroupFBErr AT %I* : BOOL;
	{attribute 'OPC.UA.DA' := '0'}
	GroupFBRun AT %I* : BOOL;
	{attribute 'OPC.UA.DA' := '0'}
	GroupInRun AT %I* : BOOL;
	{attribute 'OPC.UA.DA' := '0'}
	GroupOtherErr AT %I* : BOOL;
	{attribute 'OPC.UA.DA' := '0'}
	GroupOutErr AT %I* : BOOL;	 
	{attribute 'OPC.UA.DA' := '0'}
	GroupModuleFault AT %Q* : BOOL;
	{attribute 'OPC.UA.DA' := '0'}
	GroupStartStop AT %Q* : BOOL;
	{attribute 'OPC.UA.DA' := '0'}	
	GroupErrAck AT %Q* : BOOL;

	{attribute 'OPC.UA.DA' := '0'}
	_pulseGenerator : TON;	
	{attribute 'OPC.UA.DA' := '0'}
	_itemScheduler : INT;
	
END_VAR


IF NOT GroupInRun THEN
	IF _pulseGenerator.Q THEN
		_pulseGenerator(IN := FALSE, PT := T#10MS);
			
		CASE _itemScheduler OF					
			0:	IF NOT GroupFBRun THEN
					_logger.Information(_message.Reset().Append('Safety: started').ToString());
					GroupStartStop := TRUE;	
				END_IF
				_itemScheduler := 1;
	
			1:	IF NOT GroupErrAck THEN
					GroupErrAck := TRUE;
				END_IF
				_itemScheduler := 2;
	
			2:  IF GroupErrAck THEN
					GroupErrAck := FALSE;
					_logger.Information(_message.Reset().Append('Error acknowledgement: executed').ToString());
				END_IF
				_itemScheduler := 0;
		END_CASE
	ELSE
		_pulseGenerator(IN := TRUE, PT := T#1000MS);		
	END_IF
END_IF

END_FUNCTION_BLOCK

// ---- PMShared/Hardware/Devices/Axes/IoAxis/Stage/IoStageAxis.TcPOU
FUNCTION_BLOCK IoStageAxis EXTENDS AxesBase
VAR_INPUT
END_VAR
VAR_OUTPUT
END_VAR
VAR
	{attribute 'OPC.UA.DA' := '0'}
	_config : IoStageAxisConfig;
	{attribute 'OPC.UA.DA' := '0'}
	IoStageStruct : IoStageStruct;
	
	{attribute 'OPC.UA.DA' := '0'}
	_deliverMessages : INT;
	
	PositionMsg : STRING(255);
	
	{region 'Commands'}	
		 
	{attribute 'OPC.UA.DA' := '0'}
	_moveAbsPosition	 : BOOL;
	{attribute 'OPC.UA.DA' := '0'}			  		   
	_raiseProperties : BOOL;	 
			
	{endregion}
		 
	{attribute 'OPC.UA.DA' := '0'}
	_initDevice : BOOL;	
		
	{attribute 'OPC.UA.DA' := '0'}
	_pos : INT; //EPosition;
	{attribute 'OPC.UA.DA' := '0'}
	_itemScheduler : INT;
	{attribute 'OPC.UA.DA' := '0'}
	_itemRaisedProperties : INT;
	{attribute 'OPC.UA.DA' := '0'}
	_pulseGenerator : TON;
END_VAR


// Init device
InitDevice(); 

// Deliver messages
CASE _deliverMessages OF	
	EFeedbackMsgStage.PositionMsg :
		PositionMsg := INT_TO_STRING(GetPosition());			
END_CASE
	
_deliverMessages := 0;

// Commands
MoveAbsPosition(_moveAbsPosition, _pos); 
RaisePropertiesChanged(_raiseProperties);

IF (NOT _moveAbsPosition AND NOT _raiseProperties) THEN
	MessageScheduler();
END_IF

METHOD FB_init : BOOL
VAR_INPUT
	bInitRetains : BOOL; // if TRUE, the retain variables are initialized (warm start / cold start)
	bInCopyCode : BOOL;  // if TRUE, the instance afterwards gets moved into the copy code (online change)
	Config : IoStageAxisConfig;
END_VAR
IF Config.IsEnabled THEN
	_config := Config;
	
	SUPER^._axisConfig.Name := Config.Name;
	SUPER^._axisConfig.DeviceID := Config.DeviceID;
	SUPER^._axisConfig.IsEnabled := Config.IsEnabled;
	SUPER^._axisConfig.LogLevel := Config.LogLevel;
	
	SUPER^.Name := Config.Name;
	SUPER^.DeviceID := Config.DeviceID;	
	THIS^.Family := DeviceFamily.Axes;
	
	_Logger.Information(_message.Reset().Append('Init ').
							Append('{').Append(TO_STRING(THIS^.Family)).Append('} - ').
							Append('{').Append(TO_STRING(Config.Name)).Append('}').ToString());																													
END_IF
END_METHOD

METHOD GetPosition : INT
VAR_INPUT
END_VAR
_deliverMessages := EFeedbackMsgStage.PositionMsg;

IF IsStageInProcessPosition(IoStageStruct.InputProcessPosition) THEN
	GetPosition := EStagePosition.Process;
ELSIF IsStageInProcessPosition(IoStageStruct.InputLoadingPosition) THEN
	GetPosition := EStagePosition.Loading;
ELSE
	GetPosition := EStagePosition.Unknown;		
END_IF
END_METHOD

METHOD InitDevice : BOOL
VAR_INPUT
END_VAR
IF NOT _initDevice THEN	
	_logger.Information(_message.Reset().
								Append(_config.Name).
								Append(' - Init device').ToString());
							
	THIS^.Status := TExecutionState.Ready;
	
	GetPosition();
	
	_initDevice := TRUE;	
END_IF
END_METHOD

METHOD IsStageInLoadingPosition : BOOL
VAR_INPUT
	Position : INT;
END_VAR
VAR
	val : INT; 
END_VAR
val := ABS(Position - Const.FLEXO_AI_PISTON_LEFT_SENSING_RANGE_MAX);

IF val < Const.FLEXO_AI_PISTON_LEFT_SENSING_RANGE_MIN THEN
	IsStageInLoadingPosition := TRUE;
ELSE
	IsStageInLoadingPosition := FALSE;
END_IF
END_METHOD

METHOD IsStageInProcessPosition : BOOL
VAR_INPUT
	Position : INT;
END_VAR
VAR
	val : INT; 
END_VAR
val := ABS(Position - Const.FLEXO_AI_PISTON_LEFT_SENSING_RANGE_MAX);

IF val < Const.FLEXO_AI_PISTON_LEFT_SENSING_RANGE_MIN THEN
	IsStageInProcessPosition := TRUE;
ELSE
	IsStageInProcessPosition := FALSE;
END_IF
END_METHOD

METHOD MessageScheduler
VAR_INPUT
END_VAR
IF _pulseGenerator.Q THEN
	_pulseGenerator(IN := FALSE, PT := T#10MS);
		
	CASE _itemScheduler OF	
		0:	GetPosition();
			_itemScheduler := 0;										
	END_CASE
ELSE
	_pulseGenerator(IN := TRUE, PT := T#100MS);	
END_IF
END_METHOD

{attribute 'TcRpcEnable' := '1'}
METHOD PROTECTED MoveAbsPosition 
VAR_INPUT
	Execute : BOOL;
	Position : LREAL;
END_VAR
VAR	
END_VAR
IF Execute THEN
	_logger.Information(_message.Reset().Append(_config.Name).Append(' - Move absolute position : ').Append(TO_STRING(Position)).ToString());
	
	_moveAbsPosition := FALSE;	
	
	IF Position = EStagePosition.Loading THEN
		IoStageStruct.OutputLoadingPosition := FALSE;
		IoStageStruct.OutputProcessPosition := TRUE;		
	ELSIF Position = EStagePosition.Process THEN
		IoStageStruct.OutputLoadingPosition := TRUE;
		IoStageStruct.OutputProcessPosition := FALSE;
	ELSE
		_logger.Error(_message.Reset().Append(_config.Name).Append(' - unknown position : ').Append(TO_STRING(Position)).ToString());								
	END_IF
			
	_itemScheduler := 0;
END_IF
END_METHOD

{attribute 'TcRpcEnable' := '1'}
METHOD RaisePropertiesChanged
VAR_INPUT
	Execute : BOOL;
END_VAR
IF Execute THEN		
	_raiseProperties := TRUE;	
	
	IF _pulseGenerator.Q THEN
		_pulseGenerator(IN := FALSE, PT := T#10MS);
		
		CASE _itemRaisedProperties OF		
			0: PositionMsg := ' ';
				_itemRaisedProperties := 1;
			
			1: GetPosition();		   
				_itemRaisedProperties := 10;
				
			10: 
				_logger.Information(_message.Reset().
								    Append(_config.Name).
								    Append(' - RaisePropertiesChanged').ToString());
				_raiseProperties := FALSE;
				_itemRaisedProperties := 0;
		
		END_CASE
	
	ELSE
		_pulseGenerator(IN := TRUE, PT := T#50MS);	
	END_IF
		
END_IF
END_METHOD

METHOD ReadStagePosition
VAR_INPUT
END_VAR
END_METHOD

END_FUNCTION_BLOCK

// ---- PMShared/Hardware/Devices/Axes/AxesBase.TcPOU
FUNCTION_BLOCK ABSTRACT AxesBase EXTENDS TExecution IMPLEMENTS IDevice
VAR_INPUT
END_VAR
VAR_OUTPUT
END_VAR
VAR
	{attribute 'OPC.UA.DA' := '0'}
	_name : STRING;
	{attribute 'OPC.UA.DA' := '0'}
	_deviceID : STRING;					
	{attribute 'OPC.UA.DA' := '0'}
	_family : DeviceFamily;				
	{attribute 'OPC.UA.DA' := '0'}
	_logger : Logger;
	{attribute 'OPC.UA.DA' := '0'}
	_message : StringBuilder;	
	{attribute 'OPC.UA.DA' := '0'}
	_axisConfig : DeviceConfiguration;
	
	{attribute 'OPC.UA.DA' := '0'}
	_lifeTimeCount : UINT;
	{attribute 'OPC.UA.DA' := '0'}
	_notifyIsAlive : BOOL;
	{attribute 'OPC.UA.DA' := '0'}
	_pulseIsAliveGenerator : TON;
	
	StateMsg : STRING(255);
	IsAliveMsg : STRING(255);
END_VAR


// Check if it's still alive	
IF _notifyIsAlive THEN
	IsAliveMsg := TO_STRING(_lifeTimeCount);
	_notifyIsAlive := FALSE;
END_IF

IF HardwareGlobalVariables.ChamberState <> State THEN
	HardwareGlobalVariables.ChamberState := State;
	StateMsg := ANY_TO_STRING(State);		
END_IF

MessageScheduler();

PROPERTY DeviceID : STRING
GET
DeviceID := _deviceID;
END_GET
SET
_deviceID := DeviceID;
END_SET
END_PROPERTY

PROPERTY Family : DeviceFamily
GET
Family := _family;
END_GET
SET
_family := Family;
END_SET
END_PROPERTY

METHOD PROTECTED IsAlive
VAR_INPUT
END_VAR
_notifyIsAlive := TRUE;

IF _lifeTimeCount < 5 THEN
	_lifeTimeCount := _lifeTimeCount + 1;
ELSE
	_lifeTimeCount := 1;
END_IF
END_METHOD

METHOD MessageScheduler
VAR_INPUT
END_VAR
IF _pulseIsAliveGenerator.Q THEN
	_pulseIsAliveGenerator(IN := FALSE, PT := T#10MS);
		
	IsAlive();	
ELSE
	_pulseIsAliveGenerator(IN := TRUE, PT := T#1000MS);		
END_IF
END_METHOD

METHOD PROTECTED ABSTRACT MoveAbsPosition
VAR_INPUT
	Execute : BOOL;
	Position : LREAL; //EPosition;
END_VAR
END_METHOD

PROPERTY Name : STRING
GET
Name := _name;
END_GET
SET
_name := Name;
END_SET
END_PROPERTY

END_FUNCTION_BLOCK

// ---- PMShared/Hardware/Devices/Chambers/PSD/PsdChamber.TcPOU
 {attribute 'OPC.UA.DA' := '1'}
FUNCTION_BLOCK PsdChamber EXTENDS ChamberBase
VAR_INPUT
	IoChamberPsd : IoChamberPsd;	
END_VAR
VAR_OUTPUT
END_VAR
VAR
	{attribute 'OPC.UA.DA' := '0'}
	_config : PsdChamberConfig;
	
	{attribute 'OPC.UA.DA' := '0'}
	_initDevice : BOOL;
	
	{attribute 'OPC.UA.DA' := '0'}
	_itemInit : INT;
	{attribute 'OPC.UA.DA' := '0'}
	_itemScheduler : INT;
	{attribute 'OPC.UA.DA' := '0'}
	_itemExecScheduler : INT;		
	{attribute 'OPC.UA.DA' := '0'}
	_itemRaisedProperties : INT;			
	{attribute 'OPC.UA.DA' := '0'}
	_pulseGenerator : TON;	
	
	{region 'Commands'}	
		 	
	{attribute 'OPC.UA.DA' := '0'}
	_enableCamera : BOOL;
	{attribute 'OPC.UA.DA' := '0'}
	_moveSlitDoorPositionCmd : BOOL;
	{attribute 'OPC.UA.DA' := '0'}
	_moveCdaPneumaticValveCmd : BOOL;
	{attribute 'OPC.UA.DA' := '0'}			  		   
	_raisePropertiesCmd : BOOL;	 
			
	{endregion}
	
	{attribute 'OPC.UA.DA' := '0'}
	_deliverMessages : INT;
	
	InterlockPanelsMsg : STRING(255);	
	SlitDoorPositionMsg : STRING(255);	
	SlitDoorOpenPositionMsg : STRING(255);
	SlitDoorClosePositionMsg : STRING(255);
	CdaValveIsOpenMsg : STRING(255);
	RefreshingMsg : STRING(255);
		
	{attribute 'OPC.UA.DA' := '0'}
	message : STRING(255);
	
	{attribute 'OPC.UA.DA' := '0'}
	_pos : INT;
	{attribute 'OPC.UA.DA' := '0'}
	_openCdaValve : BOOL;
	{attribute 'OPC.UA.DA' := '0'}
	_cdaValveIsOpen : BOOL;
	
	
	{attribute 'OPC.UA.DA' := '0'}
	tmpConcat1 : STRING;
	{attribute 'OPC.UA.DA' := '0'}
	tmpConcat2 : STRING;
	{attribute 'OPC.UA.DA' := '0'}
	tmpConcatName : STRING; 
	{attribute 'OPC.UA.DA' := '0'}
	tmpConcatDescription : STRING;
	{attribute 'OPC.UA.DA' := '0'}
	tmpConcatInterlockID : STRING;
	
	{attribute 'OPC.UA.DA' := '0'}
	_itemInterlock : UINT;
	{attribute 'OPC.UA.DA' := '0'}
	_interlockCount : UINT;
		
END_VAR

SUPER^();
 
// Init device
InitDevice(); 

// Deliver messages
CASE _deliverMessages OF	
	EFeedbackMsgPsdChamber.InterlockPanelsMsg :
		InterlockPanelsMsg := message;	
	EFeedbackMsgPsdChamber.SlitDoorPositionMsg :
		SlitDoorPositionMsg := TO_STRING(SlitDoorPosition);
	EFeedbackMsgPsdChamber.SlitDoorOpenPositionMsg :
		SlitDoorOpenPositionMsg := TO_STRING(SlitDoorOpenPosition);
	EFeedbackMsgPsdChamber.SlitDoorClosePositionMsg :
		SlitDoorClosePositionMsg := TO_STRING(SlitDoorClosePosition);
	EFeedbackMsgPsdChamber.CdaValveIsOpenMsg :
		CdaValveIsOpenMsg := TO_STRING(_cdaValveIsOpen);	
END_CASE

// Commands
MoveSlitDoorPosition(_moveSlitDoorPositionCmd, _pos); 
MoveCdaPneumaticValve(_moveCdaPneumaticValveCmd, _openCdaValve); 
RaisePropertiesChanged(_raisePropertiesCmd);

IF NOT _moveSlitDoorPositionCmd AND NOT _raisePropertiesCmd THEN	
	MessageScheduler();
END_IF

PROPERTY CdaValveIsOpen : BOOL
GET
CdaValveIsOpen := _cdaValveIsOpen;
END_GET
SET
_cdaValveIsOpen := CdaValveIsOpen;
END_SET
END_PROPERTY

METHOD FB_init : BOOL
VAR_INPUT
	bInitRetains : BOOL; // if TRUE, the retain variables are initialized (warm start / cold start)
	bInCopyCode : BOOL;  // if TRUE, the instance afterwards gets moved into the copy code (online change)
	Config : PsdChamberConfig;
END_VAR
IF Config.IsEnabled THEN
	_config := Config;
	
	SUPER^._chamberConfig.Name := Config.Name;
	SUPER^._chamberConfig.DeviceID := Config.DeviceID;
	SUPER^._chamberConfig.IsEnabled := Config.IsEnabled;
	SUPER^._chamberConfig.LogLevel := Config.LogLevel;
	
	SUPER^.Name := Config.Name;
	SUPER^.DeviceID := Config.DeviceID;
	
	THIS^.Family := DeviceFamily.Chamber;

	THIS^.SetReady();
	_Logger.Information(_message.Reset().Append('Init ').
							Append('{').Append(TO_STRING(THIS^.Family)).Append('} - ').
							Append('{').Append(TO_STRING(THIS^.Name)).Append('} - ').
							Append('Status : ').Append(TO_STRING(THIS^.Status)).
							ToString());										 
END_IF
END_METHOD

METHOD InitDevice
VAR_INPUT
END_VAR
VAR	
END_VAR
IF NOT _initDevice THEN			
	_logger.Information(_message.Reset().
								Append(_config.Name).
								Append(' - init device').ToString());		
								
	IF IoChamberPsd.OutputCdaPneumaticValve = FALSE THEN
		_logger.Information(_message.Reset().Append('Start pneumatic valve').ToString());								
		IoChamberPsd.OutputCdaPneumaticValve := TRUE;
	END_IF
	
	_initDevice := TRUE;
END_IF
END_METHOD

METHOD MessageScheduler
VAR_INPUT
END_VAR
IF _pulseGenerator.Q THEN
	_pulseGenerator(IN := FALSE, PT := T#10MS);
		
	CASE _itemScheduler OF	
		0: SlitDoorPositionMsg := ' ';		   
		   CdaValveIsOpenMsg := ' ';
		   _itemScheduler := 1;
		   
		1: ReadInterlock();
		   _itemScheduler := 2;
		   
		2:  ReadSlitDoorPosition();
			_itemScheduler := 3;

		3:  ReadSlitDoorOpenPosition();
			_itemScheduler := 4;

		4:  ReadSlitDoorClosePosition();
			_itemScheduler := 5;		
					
		5:  IsReadyToLoadUnload();
			_itemScheduler := 6;	
		
		6:  ReadCdaValvePosition();
			_itemScheduler := 0;					
	END_CASE
ELSE
	_pulseGenerator(IN := TRUE, PT := T#50MS);		
END_IF
END_METHOD

{attribute 'TcRpcEnable' := '1'}
METHOD MoveCdaPneumaticValve
VAR_INPUT
	Execute : BOOL;
	OpenValve : BOOL;
END_VAR
IF Execute THEN
	_logger.Information(_message.Reset().Append(_config.Name).Append(' - Move CDA pneumatic valve : ').Append(TO_STRING(openValve)).ToString());
		
	IF OpenValve THEN
		IoChamberPsd.OutputCdaPneumaticValve := TRUE;
	ELSE
		IoChamberPsd.OutputCdaPneumaticValve := FALSE;	
	END_IF			
	
	_openCdaValve := FALSE;
END_IF
END_METHOD

{attribute 'TcRpcEnable' := '1'}
METHOD MoveSlitDoorPosition
VAR_INPUT
	Execute : BOOL;
	Position : INT;
END_VAR
IF Execute THEN
	_logger.Information(_message.Reset().Append(_config.Name).Append(' - Move slit door position : ').Append(TO_STRING(Position)).ToString());
	
	_moveSlitDoorPositionCmd := FALSE;
	
	IF Position = ESlitDoorPosition.Open THEN
		IoChamberPsd.OutputOpenSlitDoor := TRUE;
		IoChamberPsd.OutputCloseSlitDoor := FALSE;
	ELSIF Position = ESlitDoorPosition.Close THEN
		IoChamberPsd.OutputOpenSlitDoor := FALSE;
		IoChamberPsd.OutputCloseSlitDoor := TRUE;
	ELSE
		_logger.Error(_message.Reset().Append(_config.Name).Append(' - unknown position : ').Append(TO_STRING(Position)).ToString());
	END_IF
			
	_itemScheduler := 0;
END_IF
END_METHOD

{attribute 'TcRpcEnable' := '1'}
METHOD RaisePropertiesChanged
VAR_INPUT
	Execute : BOOL;
END_VAR
IF Execute THEN		
	_raisePropertiesCmd := TRUE;	
		
	IF _pulseGenerator.Q THEN
		_pulseGenerator(IN := FALSE, PT := T#10MS);
		
		CASE _itemRaisedProperties OF		
			0: 	SUPER^._raisePropertiesBase := TRUE;	
				RefreshingMsg := TO_STRING(TRUE);
				SlitDoorPositionMsg := TO_STRING(ESlitDoorPosition.Unknown);				   
				_itemRaisedProperties := 1;
			
			1:  SlitDoorOpenPositionMsg := ' ';
				_itemRaisedProperties := 2;
				
			2:	SlitDoorClosePositionMsg := ' ';
				_itemRaisedProperties := 3;
				
			3:  CdaValveIsOpenMsg := ' ';	   
				_itemRaisedProperties := 4;
				
			4:  ReadInterlock();
				_itemRaisedProperties := 5;
				
			5:  ReadInterlock();
				_itemRaisedProperties := 6;
				
			6:  ReadInterlock();
				_itemRaisedProperties := 7;
				
			7:  ReadInterlock();
				_itemRaisedProperties := 8;
				
			8:  ReadInterlock();
				_itemRaisedProperties := 9;
				
			9:  ReadInterlock();
				_itemRaisedProperties := 10;						
				
			10: RefreshingMsg := TO_STRING(FALSE);
				_itemRaisedProperties := 20;
				
			20: _logger.Information(_message.Reset().Append(_config.Name).Append(' - RaisePropertiesChanged').ToString());
				_raisePropertiesCmd := FALSE;
				_itemRaisedProperties := 0;
		END_CASE	
	ELSE
		_pulseGenerator(IN := TRUE, PT := T#100MS);	
	END_IF		
END_IF
END_METHOD

METHOD ReadCdaValvePosition 
VAR_INPUT
END_VAR
VAR
END_VAR
_deliverMessages := EFeedbackMsgPsdChamber.CdaValveIsOpenMsg;


IF IoChamberPsd.OutputCdaPneumaticValve THEN
	CdaValveIsOpen := TRUE;
ELSE
	CdaValveIsOpen := FALSE;	
END_IF
END_METHOD

METHOD ReadInterlock 
VAR_INPUT
END_VAR
VAR
	statePanel : STRING;
END_VAR
_deliverMessages := EFeedbackMsgPsdChamber.InterlockPanelsMsg;

IF _interlockCount < Const.PSD_NUMBER_INTERLOCK_PANELS THEN
	_interlockCount := _interlockCount + 1;
ELSE
	_interlockCount := 0;
END_IF

tmpConcatName := CONCAT(_config.Interlock[_interlockCount].Name, ';');
tmpConcatDescription := CONCAT(_config.Interlock[_interlockCount].Description, ';');
tmpConcatInterlockID := CONCAT(UINT_TO_STRING(_config.Interlock[_interlockCount].InterlockID), ';');

tmpConcat1 := CONCAT(tmpConcatName, tmpConcatDescription);
tmpConcat2 := CONCAT(tmpConcat1, tmpConcatInterlockID);

IF _config.Interlock[_interlockCount].State THEN
	statePanel := 'Closed';
ELSE
	statePanel := 'Open';
END_IF

message := CONCAT(tmpConcat2, statePanel);
END_METHOD

METHOD ReadSlitDoorClosePosition 
VAR_INPUT
END_VAR
VAR
	open : BOOL;
	close : BOOL;
END_VAR
_deliverMessages := EFeedbackMsgPsdChamber.SlitDoorClosePositionMsg;
SlitDoorClosePosition := IoChamberPsd.InputCloseSlitDoor;
END_METHOD

METHOD ReadSlitDoorOpenPosition 
VAR_INPUT
END_VAR
VAR
END_VAR
_deliverMessages := EFeedbackMsgPsdChamber.SlitDoorOpenPositionMsg;
SlitDoorOpenPosition := IoChamberPsd.InputOpenSlitDoor;
END_METHOD

METHOD ReadSlitDoorPosition 
VAR_INPUT
END_VAR
VAR
	open : BOOL;
	close : BOOL;
	efemOpen : BOOL;
END_VAR
_deliverMessages := EFeedbackMsgPsdChamber.SlitDoorPositionMsg;

open := IoChamberPsd.InputOpenSlitDoor;
close := IoChamberPsd.InputCloseSlitDoor;
efemOpen := IoChamberBase.InputEfemSlitDoorOpen;

IF open AND NOT close AND efemOpen THEN
	SlitDoorPosition := ESlitDoorPosition.Open;	
ELSIF close AND NOT open AND NOT efemOpen THEN
	SlitDoorPosition := ESlitDoorPosition.Close;
ELSIF close AND open THEN
	SlitDoorPosition := ESlitDoorPosition.Error;	
ELSE
	SlitDoorPosition := ESlitDoorPosition.Unknown;		
END_IF
END_METHOD

END_FUNCTION_BLOCK

// ---- PMShared/Hardware/Devices/Chucks/PSD/PsdChuck.TcPOU
FUNCTION_BLOCK PsdChuck EXTENDS ChuckBase
VAR_INPUT
	IoChuckPsd : IoChuckPsd;
END_VAR
VAR_OUTPUT
END_VAR
VAR
	{attribute 'OPC.UA.DA' := '0'}
	_config : PsdChuckConfig;
	
	{attribute 'OPC.UA.DA' := '0'}
	_deliverMessages : INT;
	
	WaferPresenceMsg : STRING(255);
	
	{attribute 'OPC.UA.DA' := '0'}
	_initDevice : BOOL;
	
	{attribute 'OPC.UA.DA' := '0'}
	_itemInit : INT;
	
	{attribute 'OPC.UA.DA' := '0'}
	_itemScheduler : INT;
	{attribute 'OPC.UA.DA' := '0'}
	_itemRaisedProperties : INT;
	{attribute 'OPC.UA.DA' := '0'}
	_pulseGenerator : TON;
	
	{region 'Commands'}
		
	{attribute 'OPC.UA.DA' := '0'}			  		   
	_raisePropertiesCmd : BOOL;
			
	{endregion}	
		
	{attribute 'OPC.UA.DA' := '0'}
	message : STRING;
	{attribute 'OPC.UA.DA' := '0'}
	_waferPresenceSensorCounter : UINT;
		 
END_VAR

SUPER^();

// Init device
InitDevice(); 

// Deliver messages
CASE _deliverMessages OF		
	EFeedbackMsgPsdChuck.WaferPresenceMsg :
		WaferPresenceMsg := message;		
END_CASE
	
_deliverMessages := 0;

// Commands	
RaisePropertiesChanged(_raisePropertiesCmd);

IF (NOT _raisePropertiesCmd) THEN
	MessageScheduler();
END_IF

METHOD FB_init : BOOL
VAR_INPUT
	bInitRetains : BOOL; // if TRUE, the retain variables are initialized (warm start / cold start)
	bInCopyCode : BOOL;  // if TRUE, the instance afterwards gets moved into the copy code (online change)
	Config : PsdChuckConfig;
END_VAR
IF Config.IsEnabled THEN
	_config := Config;
	
	SUPER^._chuckConfig.Name := Config.Name;
	SUPER^._chuckConfig.DeviceID := Config.DeviceID;
	SUPER^._chuckConfig.IsEnabled := Config.IsEnabled;
	SUPER^._chuckConfig.LogLevel := Config.LogLevel;
	
	SUPER^.Name := Config.Name;
	SUPER^.DeviceID := Config.DeviceID;
	
	THIS^.Family := DeviceFamily.Chuck;

	THIS^.SetReady();
	_Logger.Information(_message.Reset().Append('Init ').
							Append('{').Append(TO_STRING(THIS^.Family)).Append('} - ').
							Append('{').Append(TO_STRING(THIS^.Name)).Append('} - ').
							Append('Status : ').Append(TO_STRING(THIS^.Status)).
							ToString());										 
END_IF
END_METHOD

METHOD InitDevice
VAR_INPUT
END_VAR
IF NOT _initDevice THEN			
	_logger.Information(_message.Reset().
								Append(_config.Name).
								Append(' - init device').ToString());		
								
	_initDevice := TRUE;
END_IF
END_METHOD

METHOD MessageScheduler
VAR_INPUT
END_VAR
IF _pulseGenerator.Q THEN
	_pulseGenerator(IN := FALSE, PT := T#10MS);
		
	CASE _itemScheduler OF	
		0:	WaferPresenceMsg := ' ';
			_itemScheduler := 1;
	
		1:	ReadWaferPresence();
			_itemScheduler := 0;		
									
	END_CASE
ELSE
	_pulseGenerator(IN := TRUE, PT := T#100MS);	
END_IF
END_METHOD

{attribute 'TcRpcEnable' := '1'}
METHOD RaisePropertiesChanged
VAR_INPUT
	Execute : BOOL;
END_VAR
VAR	
	waferPresence : STRING;
	diameter : STRING;
END_VAR
IF Execute THEN		
	_raisePropertiesCmd := TRUE;	
	
	IF _pulseGenerator.Q THEN
		_pulseGenerator(IN := FALSE, PT := T#10MS);
		
		CASE _itemRaisedProperties OF		
			0:  diameter := TO_STRING(_config.WaferPresenceSensor[_waferPresenceSensorCounter].Diameter);
				WaferPresenceMsg := CONCAT(CONCAT(diameter, ';'), INT_TO_STRING(EMaterialPresence.Unknown));
				_itemRaisedProperties := 10;
				
			10: _logger.Information(_message.Reset().Append(_config.Name).Append(' - RaisePropertiesChanged').ToString());
				_raisePropertiesCmd := FALSE;
				_itemRaisedProperties := 0;		
		END_CASE	
	ELSE
		_pulseGenerator(IN := TRUE, PT := T#100MS);	
	END_IF		
END_IF
END_METHOD

METHOD ReadWaferPresence
VAR_INPUT
END_VAR
VAR	
	waferPresence : STRING;
	diameter : STRING;
END_VAR
_deliverMessages := EFeedbackMsgPsdChuck.WaferPresenceMsg;

IF _waferPresenceSensorCounter < Const.PSD_NUMBER_WAFER_PRESENCE_SENSORS - 1 THEN
	_waferPresenceSensorCounter := _waferPresenceSensorCounter + 1;
ELSE
	_waferPresenceSensorCounter := 0;
END_IF

diameter := TO_STRING(_config.WaferPresenceSensor[_waferPresenceSensorCounter].Diameter);
IF _config.WaferPresenceSensor[_waferPresenceSensorCounter].InputWaferPresence THEN
	waferPresence := INT_TO_STRING(EMaterialPresence.Present);
ELSE
	waferPresence := INT_TO_STRING(EMaterialPresence.NotPresent);		
END_IF

message := CONCAT(CONCAT(diameter, ';'), waferPresence);
END_METHOD

END_FUNCTION_BLOCK

// ---- PMShared/Hardware/Devices/Chucks/ChuckBase.TcPOU
FUNCTION_BLOCK ABSTRACT ChuckBase EXTENDS TExecution IMPLEMENTS IDevice
VAR_INPUT
END_VAR
VAR_OUTPUT
END_VAR
VAR
	{attribute 'OPC.UA.DA' := '0'}
	_name : STRING;
	{attribute 'OPC.UA.DA' := '0'}
	_deviceID : STRING;				
	{attribute 'OPC.UA.DA' := '0'}
	_family : DeviceFamily := DeviceFamily.Chuck;		
	{attribute 'OPC.UA.DA' := '0'}
	_logger : Logger;
	{attribute 'OPC.UA.DA' := '0'}
	_message : StringBuilder;
	{attribute 'OPC.UA.DA' := '0'}
	_chuckConfig : DeviceConfiguration;
	
	{attribute 'OPC.UA.DA' := '0'}
	_lifeTimeCount : UINT;
	{attribute 'OPC.UA.DA' := '0'}
	_notifyIsAlive : BOOL;
	{attribute 'OPC.UA.DA' := '0'}
	_pulseIsAliveGenerator : TON;
	{attribute 'OPC.UA.DA' := '0'}
	_pulseGeneratorBase : TON;
	{attribute 'OPC.UA.DA' := '0'}
	_execPulseGeneratorBase : TON;	
	
	{attribute 'OPC.UA.DA' := '0'}
	_itemSchedulerBase : INT;
	{attribute 'OPC.UA.DA' := '0'}
	_itemExecSchedulerBase : INT;	
	
	{attribute 'OPC.UA.DA' := '0'}
	_deliverMessagesBase : INT;
	
	{attribute 'OPC.UA.DA' := '0'}
	_chuckInLoadingPositionCmd : BOOL;
	
	StateMsg : STRING(255);
	IsAliveMsg : STRING(255);
	IsInLoadingPositionMsg : STRING(255);
	
	{attribute 'OPC.UA.DA' := '0'}
	_isInLoadingPosition : BOOL;
	{attribute 'OPC.UA.DA' := '0'}
	_loadingPosition : BOOL;		
	{attribute 'OPC.UA.DA' := '0'}
	IsInLoadingPosition AT %Q* : BOOL;
	
	{attribute 'OPC.UA.DA' := '0'}	
	_waferSize : EWaferSize := EWaferSize.Unknown; 
	
	{attribute 'OPC.UA.DA' := '0'}
	ioMessage : STRING;
END_VAR

// Check if it's still alive	
IF _notifyIsAlive THEN
	IsAliveMsg := TO_STRING(_lifeTimeCount);
	_notifyIsAlive := FALSE;
END_IF

IF HardwareGlobalVariables.ChuckState <> State THEN
	HardwareGlobalVariables.ChuckState := State;
	StateMsg := ANY_TO_STRING(State);		
END_IF

CASE _deliverMessagesBase OF		
	EFeedbackMsgChuckBase.IsInLoadingPositionMsg :	
		IsInLoadingPositionMsg := ioMessage;		
END_CASE

ChuckInLoadingPosition(_chuckInLoadingPositionCmd, _loadingPosition);

IF NOT _chuckInLoadingPositionCmd THEN
	MessageSchedulerBase();	
END_IF

{attribute 'TcRpcEnable' := '1'}
METHOD ChuckInLoadingPosition
VAR_INPUT
	Execute : BOOL;
	LoadingPosition : BOOL;
END_VAR

